REGION Network 13: Special characters — Arrows, box and block characters
   // ▄▄▄▄▄▄▄▄▄▄▄▄▄▄▄▄▄▄▄▄▄▄▄▄▄▄▄▄▄▄▄▄▄▄▄▄▄▄▄▄▄▄▄▄
   // ARROWS
   // 
   // 
   // ← Left Arrow              ⇐ Left dbl Arrow             ↩ Left Arrow Hook
   // ↑ Up Arrow               ⇑ Up dbl Arrow               ↪ Right Arrow Hook
   // → Right Arrow              ⇒ Right dbl Arrow           ⤣ North West Arrow Hook
   // ↓ Down Arrow             ⇓ Down dbl Arrow             ⤤ North East Arrow Hook
   // ↔ Left Right Arrow             ⇔ Left Right dbl Arrow          ⤥ South East Arrow Hook
   // ↕ Up Down Arrow          ⇕ Up Down dbl Arrow          ⤦ South West Arrow Hook
   // ↖ North West Arrow          ⇖ North West dbl Arrow         ↰    Up Arrow Tip Left
   // ↗ North East Arrow          ⇗ North East dbl Arrow          ↱    Up Arrow Tip Right
   // ↘ South East Arrow          ⇘ South East dbl Arrow         ↲    Down Arrow Tip Left
   // ↙ South West Arrow         ⇙    South West dbl Arrow        ↳ Down Arrow Tip Right
   // ⤡ North West & South East Arrow    ⤂ Left dbl Arrow vert Stroke       ↴ Right Arrow Corner down
   // ⤢ North East & South West Arrow    ⤃ Right dbl Arrow vert Stroke     ↵ Down Arrow Corner Left
   // ⇄ Right Arrow Over Left Arrow       ⤆ Left dbl Arrow From Bar        ↶ Anticlockwise Top Semicircle Arrow
   // ⇅ Up Arrow Left Of down Arrow        ⤇ Right dbl Arrow From Bar         ↷ Clockwise Top Semicircle Arrow
   // ⇆ Left Arrow Over Right Arrow       ⤄ Left Right dbl Arrow vert Stroke    ↺ Anticlockwise Open Circle Arrow
   // ⇇ Left Paired Arrows           ↼ Left Harpoon Barb up         ↻ Clockwise Open Circle Arrow
   // ⇈ Up Paired Arrows             ↽ Left Harpoon Barb down         ⟲ Anticlockwise Gapped Circle Arrow
   // ⇉ Right Paired Arrows         ↾ Up Harpoon Barb Right         ⟳ Clockwise Gapped Circle Arrow
   // ⇊ Down Paired Arrows           ↿ Up Harpoon Barb Left
   // ↤ Left Arrow From Bar           ⇀ Right Harpoon Barb up         ▲  Black Up Triangle 
   // ↥ Up Arrow From Bar          ⇁ Right Harpoon Barb down       ▼  Black Down Triangle
   // ↦ Right Arrow From Bar         ⇂ Down Harpoon Barb Right      ▶  Black Right Triangle
   // ↧ down Arrow From Bar        ⇃ Down Harpoon Barb Left         ◀  Black Left Triangle
   // ↨ Up Down Arrow Base         ⇋ Left Harpoon Over Right Harpoon
   // ↞ Left Two head Arrow          ⇌ Right Harpoon Over Left Harpoon
   // ↟ up Two head Arrow         ↯ Down Zigzag Arrow
   // ↠ Right Two head Arrow
   // ↡ Down Two head Arrow
   // ⤙ Left Arrow-Tail
   // ⤚ Right Arrow-Tail
   // ⤛ Left dbl Arrow-Tail    
   // ⤜ Right dbl Arrow-Tail    
   // ⤝ Left Arrow To Black Diamond    
   // ⤞ Right Arrow To Black Diamond    
   // 
   // ⟵  Long Left Arrow             ↢ Left Arrow Tail             ⌃   Up Arrowhead
   // ⟶  Long Right Arrow          ↣ Right Arrow Tail             ⌄   Down Arrowhead
   // ⟷  Long Left Right Arrow         ⤟ Left Arrow Bar To Black Diamond   ⌅   Projective
   // ⟸  Long Left dbl Arrow         ⤠ Right Arrow Bar To Black Diamond    ⌆   Perspective
   // ⟹  Long Right dbl Arrow          ⤌    Left dbl Dash Arrow         ⟰ Up Quadruple Arrow
   // ⟺  Long Left Right dbl Arrow        ⤍    Right dbl Dash Arrow         ⟱ Down Quadruple Arrow
   // ⟻  Long Left Arrow From Bar       ⤎    Left Triple Dash Arrow        ⤊ Up Triple Arrow
   // ⟼  Long Right Arrow From Bar        ⤏    Right Triple Dash Arrow         ⤋ Down Triple Arrow
   // ⟽  Long Left dbl Arrow From Bar       ⤈    Down Arrow horiz Stroke          ⤈   Down Arrow horiz Stroke
   // ⟾  Long Right dbl Arrow From Bar    ⤉    Up Arrow horiz Stroke             ⤉   Up Arrow horiz Stroke
   // 
   // 
   // 
   // ▄▄▄▄▄▄▄▄▄▄▄▄▄▄▄▄▄▄▄▄▄▄▄▄▄▄▄▄▄▄▄▄▄▄▄▄▄▄▄▄▄▄▄▄
   // BOX CHARACTERS
   // 
   // 
   // ─ Box Light horiz            ╌ Box Light dbl Dash horiz       ⋮     Vert Ellipsis
   // │ Box Light vert             ╎ Box Light dbl Dash vert        ⋯    Midline horiz Ellipsis
   // ╱ Box Light diag top Right Left      ╍ Box Heavy dbl Dash horiz       ⋰     Up Right diag Ellipsis
   // ╲ Box Light diag top Left To btm Right    ╏ Box Heavy dbl Dash vert          ⋱    Down Right diag Ellipsis
   // ╳ Box Light diag Cross          ┄ Box Light Triple Dash horiz      ╴ Box Light Left
   // ━ Box Heavy horiz             ┆ Box Light Triple Dash vert       ╵ Box Light Up
   // ┃ Box Heavy vert           ┅ Box Heavy Triple Dash horiz       ╶ Box Light Right
   // ═ Box dbl horiz               ┇ Box Heavy Triple Dash vert        ╷ Box Light Down
   // ║ Box dbl vert              ┈ Box Light Quadruple Dash horiz     ╸ Box Heavy Left
   //                       ┊ Box Light Quadruple Dash vert       ╹ Box Heavy Up
   //                       ┉ Box Heavy Quadruple Dash horiz      ╺ Box Heavy Right
   //                       ┋ Box Heavy Quadruple Dash vert     ╻ Box Heavy Down
   // 
   // ┌ Box Light Down & Right        ├ Box Light vert & Right         ─ Box Light horiz
   // └ Box Light Up & Right           ┤ Box Light vert & Left        │ Box Light vert
   // ┐ Box Light Down & Left           ┬ Box Light Down & horiz         ┼ Box Light vert & horiz
   // ┘ Box Light Up & Left          ┴ Box Light Up & horiz  
   // ┏ Box Heavy Down & Right         ┣ Box Heavy vert & Right          ━ Box Heavy horiz
   // ┗ Box Heavy Up & Right         ┫ Box Heavy vert & Left         ┃ Box Heavy vert
   // ┓ Box Heavy Down & Left         ┳ Box Heavy Down & horiz       ╋ Box Heavy vert & horiz
   // ┛ Box Heavy Up & Left        ┻ Box Heavy Up & horiz  
   //     
   // ┍ Box Down Light & Right Heavy     ┝ Box vert Light & Right Heavy      ━ Box Heavy horiz
   // ┕ Box Up Light & Right Heavy        ┥ Box vert Light & Left Heavy     │ Box Light vert
   // ┑ Box Down Light & Left Heavy     ┯ Box Down Light & horiz Heavy      ┿ Box vert Light & horiz Heavy
   // ┙ Box Up Light & Left Heavy       ┷ Box Up Light & horiz Heavy  
   // 
   // ┎ Box Down Heavy & Right Light     ┠ Box vert Heavy & Right Light      ─ Box Light horiz
   // ┖ Box Up Heavy & Right Light        ┨ Box vert Heavy & Left Light     ┃ Box Heavy vert
   // ┒ Box Down Heavy & Left Light     ┰ Box Down Heavy & horiz Light      ╂ Box vert Heavy & horiz Light
   // ┚ Box Up Heavy & Left Light       ┸ Box Up Heavy & horiz Light  
   // 
   // ┦ Box Up Heavy & Left Down Light     ┪ Box Up Light & Left Down Heavy     ╀ Box Up Heavy & Down horiz Light
   // ┶ Box Right Heavy & Left Up Light   ┹ Box Right Light & Left Up Heavy   ┾ Box Right Heavy & Left vert Light
   // ┟ Box Down Heavy & Right Up Light     ┡ Box Down Light & Right Up Heavy     ╁ Box Down Heavy & Up horiz Light
   // ┭ Box Left Heavy & Right Down Light    ┲ Box Left Light & Right Down Heavy    ┽ Box Left Heavy & Right vert Light
   //  
   // ┞ Box Up Heavy & Right Down Light     ┢ Box Up Light & Right Down Heavy     ╈ Box Up Light & Down horiz Heavy
   // ┮ Box Right Heavy & Left Down Light    ┱ Box Right Light & Left Down Heavy    ╉ Box Right Light & Left vert Heavy
   // ┧ Box Down Heavy & Left Up Light     ┩ Box Down Light & Left Up Heavy     ╇ Box Down Light & Up horiz Heavy
   // ┵ Box Left Heavy & Right Up Light      ┺ Box Left Light & Right Up Heavy   ╊ Box Left Light & Right vert Heavy
   // 
   // ╼ Box Light Left & Heavy Right                            ╄ Box Right Up Heavy & Left Down Light
   // ╽ Box Light Up & Heavy Down                            ╆ Box Right Down Heavy & Left Up Light
   // ╾ Box Heavy Left & Light Right                            ╅ Box Left Down Heavy & Right Up Light
   // ╿ Box Heavy Up & Light Down                            ╃ Box Left Up Heavy & Right Down Light
   // 
   // ╔ Box dbl Down & Right         ╠ Box dbl vert & Right         ═ Box dbl horiz
   // ╚ Box dbl Up & Right           ╣ Box dbl vert & Left           ║ Box dbl vert
   // ╗ Box dbl Down & Left        ╦ Box dbl Down & horiz         ╬ Box dbl vert & horiz
   // ╝ Box dbl Up & Left          ╩ Box dbl Up & horiz  
   //  
   // ╒ Box Down Single & Right dbl     ╞ Box vert Single & Right dbl      ═ Box dbl horiz
   // ╘ Box Up Single & Right dbl        ╡ Box vert Single & Left dbl        │ Box Light vert
   // ╕ Box Down Single & Left dbl        ╤ Box Down Single & horiz dbl      ╪ Box vert Single & horiz dbl
   // ╛ Box Up Single & Left dbl       ╧ Box Up Single & horiz dbl  
   // 
   // ╓ Box Down dbl & Right Single     ╟ Box vert dbl & Right Single      ─ Box Light horiz
   // ╙ Box Up dbl & Right Single        ╢ Box vert dbl & Left Single        ║ Box dbl vert
   // ╖ Box Down dbl & Left Single        ╥ Box Down dbl & horiz Single      ╫ Box vert dbl & horiz Single
   // ╜ Box Up dbl & Left Single       ╨ Box Up dbl & horiz Single  
   // 
   // 
   // 
   // ▄▄▄▄▄▄▄▄▄▄▄▄▄▄▄▄▄▄▄▄▄▄▄▄▄▄▄▄▄▄▄▄▄▄▄▄▄▄▄▄▄▄▄▄
   // BLOCK CHARACTERS
   // 
   // 
   // ▀ Top Half Block             ❘    Light vert Bar              ❘ ❘     En Space
   // ▄ Btm Half Block            ❙    Medium vert Bar           ❘ ❘   Em Space
   // ▐ Right Half Block          ❚   Heavy vert Bar  
   // ▌ Left Half Block    
   // 
   // ▔ Top One Eighth Block        ▉ Left Seven Eighths Block
   // ▁ Btm One Eighth Block          ▊ Left Three Quarters Block
   // ▂ Btm One Quarter Block        ▋ Left Five Eighths Block
   // ▃ Btm Three Eighths Block      ▌ Left Half Block
   // ▄ Btm Half Block            ▍ Left Three Eighths Block
   // ▅ Btm Five Eighths Block         ▎ Left One Quarter Block
   // ▆ Btm Three Quarters Block       ▏ Left One Eighth Block
   // ▇ Btm Seven Eighths Block        ▕ Right One Eighth Block
   // █ Full Block
   // ░ Light Shade
   // ▒ Medium Shade    
   // ▓ Dark Shade    
   // 
   // 
   // ██████████████ █ █ █ █  END   █ █ █ █ ██████████████
END_REGION

REGION Network 14: Special characters — Currency, punctuation and full-width characters
   // ▄▄▄▄▄▄▄▄▄▄▄▄▄▄▄▄▄▄▄▄▄▄▄▄▄▄▄▄▄▄▄▄▄▄▄▄▄▄▄▄▄▄▄▄
   // CURRENCY
   // 
   // 
   // ₳   Austral Sign             €   Euro Sign              ₦  Naira Sign
   // ₵   Cedi Sign               ₠  Euro-Currency Sign          ₪  New Shekel Sign
   // ¢   Cent Sign              ₣  French Franc Sign           ₧   Peseta Sign
   // ₡   Colon Sign               ₰   German Penny Sign           ₱   Peso Sign
   // ₢   Cruzeiro Sign           ₲   Guarani Sign              £  Pound Sign
   // ¤  Currency Sign             ₴   Hryvnia Sign            ₨    Rupee Sign
   // $   Dollar Sign            ₭   Kip Sign              ₮   Tugrik Sign
   // ₫   Dong Sign             ₤   Lira Sign             ₩  Won Sign
   // ₯ Drachma Sign            ₥  Mill Sign              ¥   Yen Sign
   // 
   // 
   // 
   // ▄▄▄▄▄▄▄▄▄▄▄▄▄▄▄▄▄▄▄▄▄▄▄▄▄▄▄▄▄▄▄▄▄▄▄▄▄▄▄▄▄▄▄▄
   // PUNCTUATION AND COMMON SYMBOLS
   // 
   // 
   // #  Hash Sign             "   Quote                 §   Section Sign
   // $   Dollar Sign            “    Left dbl quote             ¶   Pilcrow Sign
   // %  Percent Sign            ”    Right dbl quote
   // &   Ampersand             '    Apostrophe  
   // *   Asterisk              ‘    Left Single quote          †   Dagger
   // ~   Tilde                 ’    Right Single quote           ‡   Dbl Dagger
   // +   Plus Sign               ‹    Single Left Angle quote       •   Bullet
   // -    Hyphen/minus            ›    Single Right Angle quote        ·    Middle Dot
   // =   Equals Sign                                ‣   Triangular Bullet
   // <   Less-Than Sign           ´   Acute Accent              ⁃    Hyphen Bullet
   // >   Greater-Than Sign           `   Grave Accent
   // (    Left Parenthesis
   // )    Right Parenthesis            ©  Copyright Sign           ⁎   Low Asterisk
   // [    Left Square Bracket           ®  Registered Sign  
   // ]    Right Square Bracket         ℀  Account Of               ․    One Dot Leader
   // {   Left Curly Bracket          ℁  Addressed To The Subject      ‥   Two Dot Leader
   // }   Right Curly Bracket          ℂ  Dbl-Struck Capital C           …  Horiz Ellipsis
   // 〈    Left Angle Bracket           ℄   Centre Line Symbol  
   // 〉    Right Angle Bracket            ℅  Care Of               ※  Reference Mark
   // ⁅    Left Square Bracket Quill        ℗  Sound Recording Copyright       ‼   Dbl Exclamation Mark
   // ⁆    Right Square Bracket Quill      ™  Trade Mark Sign            ‽   Interrobang
   // ,    Comma                                 ⁇  Dbl Question Mark
   // .    Full Stop                                   ⁈   Question Exclamation Mark
   // :    Colon                                  ⁉  Exclamation Question Mark
   // ;    Semicolon    
   // !    Exclamation Mark            ⁑   Two Asterisks Aligned vertically     |    Vert Line
   // ?   Question Mark           ⁂   Asterism               ¦    Broken Bar
   // @  Commercial At                              ‖    Dbl vert Line
   // ^   Circumflex Accent            ⁀  Character Tie              ‗   Dbl Low Line
   // /    Solidus               ‿  Undertie             ⁞    Vert Four Dots
   // \    Reverse Solidus            ⁐  Close Up
   // _   Underscore
   // ― Horiz Bar    
   // ¯   Macron
   // ‾   Overline
   // 
   // 
   // 
   // ▄▄▄▄▄▄▄▄▄▄▄▄▄▄▄▄▄▄▄▄▄▄▄▄▄▄▄▄▄▄▄▄▄▄▄▄▄▄▄▄▄▄▄▄
   // NON-PROPORTIONAL (FULL-WIDTH) LETTERS
   // 
   // 
   // Ａ Fullwidth Capital Letter A        ａ Fullwidth Small Letter A       ＂ Fullwidth quote
   // Ｂ Fullwidth Capital Letter B        ｂ Fullwidth Small Letter B       ＇ Fullwidth Apostrophe
   // Ｃ Fullwidth Capital Letter C        ｃ Fullwidth Small Letter C       ＃ Fullwidth Number Sign
   // Ｄ Fullwidth Capital Letter D       ｄ Fullwidth Small Letter D       ＄ Fullwidth Dollar Sign
   // Ｅ Fullwidth Capital Letter E        ｅ Fullwidth Small Letter E       ％ Fullwidth Percent Sign
   // Ｆ Fullwidth Capital Letter F        ｆ Fullwidth Small Letter F       ＆ Fullwidth Ampers&
   // Ｇ Fullwidth Capital Letter G       ｇ Fullwidth Small Letter G       ＊ Fullwidth Asterisk
   // Ｈ Fullwidth Capital Letter H       ｈ Fullwidth Small Letter H          ～ Fullwidth Tilde
   // Ｉ Fullwidth Capital Letter I         ｉ Fullwidth Small Letter I        ＋ Fullwidth Plus Sign
   // Ｊ Fullwidth Capital Letter J         ｊ Fullwidth Small Letter J        － Fullwidth Hyphen-Minus
   // Ｋ Fullwidth Capital Letter K        ｋ Fullwidth Small Letter K       ＝ Fullwidth Equals Sign
   // Ｌ Fullwidth Capital Letter L        ｌ Fullwidth Small Letter L       ＜ Fullwidth Less-Than Sign
   // Ｍ Fullwidth Capital Letter M       ｍ Fullwidth Small Letter M         ＞ Fullwidth Greater-Than Sign
   // Ｎ Fullwidth Capital Letter N       ｎ Fullwidth Small Letter N          （ Fullwidth Left Parenthesis
   // Ｏ Fullwidth Capital Letter O       ｏ Fullwidth Small Letter O       ） Fullwidth Right Parenthesis
   // Ｐ Fullwidth Capital Letter P        ｐ Fullwidth Small Letter P       ［ Fullwidth Left Square Bracket
   // Ｑ Fullwidth Capital Letter Q       ｑ Fullwidth Small Letter Q         ］ Fullwidth Right Square Bracket
   // Ｒ Fullwidth Capital Letter R        ｒ Fullwidth Small Letter R       ｛ Fullwidth Left Curly Bracket
   // Ｓ Fullwidth Capital Letter S        ｓ Fullwidth Small Letter S       ｝ Fullwidth Right Curly Bracket
   // Ｔ Fullwidth Capital Letter T        ｔ Fullwidth Small Letter T        ， Fullwidth Comma
   // Ｕ Fullwidth Capital Letter U       ｕ Fullwidth Small Letter U       ． Fullwidth Full Stop
   // Ｖ Fullwidth Capital Letter V        ｖ Fullwidth Small Letter V       ： Fullwidth Colon
   // Ｗ Fullwidth Capital Letter W       ｗ Fullwidth Small Letter W         ； Fullwidth Semicolon
   // Ｘ Fullwidth Capital Letter X        ｘ Fullwidth Small Letter X       ！ Fullwidth Exclamation Mark
   // Ｙ Fullwidth Capital Letter Y        ｙ Fullwidth Small Letter Y       ？ Fullwidth Question Mark
   // Ｚ Fullwidth Capital Letter Z        ｚ Fullwidth Small Letter Z       ＠ Fullwidth Commercial At
   //                                         ＾ Fullwidth Circumflex Accent
   // ０ Fullwidth Digit Zero         ５ Fullwidth Digit Five          ／ Fullwidth Solidus
   // １ Fullwidth Digit One         ６ Fullwidth Digit Six         ＼ Fullwidth Reverse Solidus
   // ２ Fullwidth Digit Two          ７ Fullwidth Digit Seven         ＿ Fullwidth Low Line
   // ３ Fullwidth Digit Three          ８ Fullwidth Digit Eight           ｜ Fullwidth vert Line
   // ４ Fullwidth Digit Four         ９ Fullwidth Digit Nine         ❘ ❘   Fullwidth space    
   // 
   // 
   // ██████████████ █ █ █ █  END   █ █ █ █ ██████████████
END_REGION

REGION Network 15: Special characters — Greek, indexing characters and Roman numerals
   // ▄▄▄▄▄▄▄▄▄▄▄▄▄▄▄▄▄▄▄▄▄▄▄▄▄▄▄▄▄▄▄▄▄▄▄▄▄▄▄▄▄▄▄▄
   // GREEK CHARACTERS
   // 
   // 
   // Α  Greek Capital Letter Alpha        α   Greek Small Letter Alpha
   // Β   Greek Capital Letter Beta       β   Greek Small Letter Beta
   // Γ   Greek Capital Letter Gamma       γ   Greek Small Letter Gamma
   // Δ  Greek Capital Letter Delta      δ   Greek Small Letter Delta
   // Ε   Greek Capital Letter Epsilon     ε   Greek Small Letter Epsilon
   // Ζ   Greek Capital Letter Zeta       ζ   Greek Small Letter Zeta
   // Η  Greek Capital Letter Eta       η   Greek Small Letter Eta
   // Θ  Greek Capital Letter Theta      θ   Greek Small Letter Theta
   // Ι    Greek Capital Letter Iota         ι    Greek Small Letter Iota
   // Κ   Greek Capital Letter Kappa       κ   Greek Small Letter Kappa
   // Λ   Greek Capital Letter Lambda       λ   Greek Small Letter Lambda
   // Μ  Greek Capital Letter Mu       μ   Greek Small Letter Mu
   // Ν  Greek Capital Letter Nu        ν   Greek Small Letter Nu
   // Ξ   Greek Capital Letter Xi         ξ   Greek Small Letter Xi
   // Ο  Greek Capital Letter Omicron      ο   Greek Small Letter Omicron
   // Π  Greek Capital Letter Pi          π   Greek Small Letter Pi
   // Ρ   Greek Capital Letter Rho      ρ   Greek Small Letter Rho
   // Σ   Greek Capital Letter Sigma       ς   Greek Small Letter Final Sigma
   //                       σ   Greek Small Letter Sigma
   // Τ   Greek Capital Letter Tau         τ   Greek Small Letter Tau
   // Υ   Greek Capital Letter Upsilon     υ   Greek Small Letter Upsilon
   // Φ  Greek Capital Letter Phi       φ  Greek Small Letter Phi
   // Χ   Greek Capital Letter Chi       χ   Greek Small Letter Chi
   // Ψ  Greek Capital Letter Psi        ψ  Greek Small Letter Psi
   // 
   // 
   // 
   // ▄▄▄▄▄▄▄▄▄▄▄▄▄▄▄▄▄▄▄▄▄▄▄▄▄▄▄▄▄▄▄▄▄▄▄▄▄▄▄▄▄▄▄▄
   // INDEXING CHARACTERS  (all characters are 1 EM wide)
   // 
   // 
   // ① Circled One              ⑴ Bracketed One           ⒈ One Full Stop
   // ② Circled Two              ⑵ Bracketed Two           ⒉ Two Full Stop
   // ③ Circled Three              ⑶ Bracketed Three           ⒊ Three Full Stop
   // ④ Circled Four             ⑷ Bracketed Four             ⒋ Four Full Stop
   // ⑤ Circled Five              ⑸ Bracketed Five           ⒌ Five Full Stop
   // ⑥ Circled Six             ⑹ Bracketed Six             ⒍ Six Full Stop
   // ⑦ Circled Seven             ⑺ Bracketed Seven          ⒎ Seven Full Stop
   // ⑧ Circled Eight            ⑻ Bracketed Eight            ⒏ Eight Full Stop
   // ⑨ Circled Nine             ⑼ Bracketed Nine          ⒐ Nine Full Stop
   // ⑩ Circled Ten            ⑽ Bracketed Ten            ⒑ Ten Full Stop
   // ⑪ Circled Eleven            ⑾ Bracketed Eleven         ⒒ Eleven Full Stop
   // ⑫ Circled Twelve            ⑿ Bracketed Twelve         ⒓ Twelve Full Stop
   // ⑬ Circled Thirteen             ⒀ Bracketed Thirteen          ⒔ Thirteen Full Stop
   // ⑭ Circled Fourteen           ⒁ Bracketed Fourteen        ⒕ Fourteen Full Stop
   // ⑮ Circled Fifteen            ⒂ Bracketed Fifteen         ⒖ Fifteen Full Stop
   // ⑯ Circled Sixteen           ⒃ Bracketed Sixteen           ⒗ Sixteen Full Stop
   // ⑰ Circled Seventeen           ⒄ Bracketed Seventeen        ⒘ Seventeen Full Stop
   // ⑱ Circled Eighteen           ⒅ Bracketed Eighteen        ⒙ Eighteen Full Stop
   // ⑲ Circled Nineteen           ⒆ Bracketed Nineteen           ⒚ Nineteen Full Stop
   // ⑳ Circled Twenty            ⒇ Bracketed Twenty         ⒛ Twenty Full Stop
   // 
   // 
   // 
   // ▄▄▄▄▄▄▄▄▄▄▄▄▄▄▄▄▄▄▄▄▄▄▄▄▄▄▄▄▄▄▄▄▄▄▄▄▄▄▄▄▄▄▄▄
   // ROMAN NUMERALS
   // 
   // 
   // Ⅰ    Roman num One          ⅰ    Small Roman num One
   // Ⅱ   Roman num Two           ⅱ   Small Roman num Two
   // Ⅲ  Roman num Three           ⅲ  Small Roman num Three
   // Ⅳ  Roman num Four          ⅳ  Small Roman num Four
   // Ⅴ   Roman num Five          ⅴ   Small Roman num Five
   // Ⅵ  Roman num Six             ⅵ  Small Roman num Six
   // Ⅶ Roman num Seven         ⅶ    Small Roman num Seven
   // Ⅷ    Roman num Eight           ⅷ   Small Roman num Eight
   // Ⅸ  Roman num Nine            ⅸ  Small Roman num Nine
   // Ⅹ   Roman num Ten           ⅹ   Small Roman num Ten
   // Ⅺ  Roman num Eleven           ⅺ  Small Roman num Eleven
   // Ⅻ Roman num Twelve           ⅻ  Small Roman num Twelve
   // Ⅼ   Roman num Fifty           ⅼ    Small Roman num Fifty
   // Ⅽ   Roman num One Hundred        ⅽ   Small Roman num One Hundred
   // Ⅾ  Roman num Five Hundred      ⅾ   Small Roman num Five Hundred
   // Ⅿ  Roman num One Thousand      ⅿ     Small Roman num One Thousand    
   // 
   // 
   // ████████████████████ END    ████████████████████
END_REGION

REGION Network 16: Special characters — Mathematical operators (including vulgar fractions)
   // ▄▄▄▄▄▄▄▄▄▄▄▄▄▄▄▄▄▄▄▄▄▄▄▄▄▄▄▄▄▄▄▄▄▄▄▄▄▄▄▄▄▄▄▄
   // MATHEMATICAL OPERATORS
   // 
   // 
   // ×   Multiplication Sign          ¹   Superscript One           ∅  Empty Set
   // ÷   Division Sign              ²   Superscript Two            ∈  Element Of
   // +   Plus sign                ³   Superscript Three         ∉  Not An Element Of
   // −   Minus Sign            ½  Vulgar Fraction One Half         ∊   Small Element Of
   // ⁒   Commercial Minus Sign       ⅓  Vulgar Fraction One Third       ∋  Contains As Member
   // ±   Plus-Minus Sign             ⅔  Vulgar Fraction Two Thirds      ∌  Does Not Contain As Member
   // ∓   Minus-Or-Plus Sign          ¼  Vulgar Fraction One Quarter        ∍   Small Contains As Member
   // ≤   Less-Than Or Equal To       ¾  Vulgar Fraction Three Quarters      ∩   Intersection
   // ≥   Greater-Than Or Equal To        ⅕  Vulgar Fraction One Fifth        ∪   Union
   // ≪  Much Less-Than            ⅖  Vulgar Fraction Two Fifths       ⊂  Subset Of
   // ≫  Much Greater-Than          ⅗  Vulgar Fraction Three Fifths       ⊃  Superset Of
   // √  Square Root             ⅘  Vulgar Fraction Four Fifths      ⊄  Not A Subset Of
   // ∛  Cube Root             ⅙  Vulgar Fraction One Sixth       ⊅  Not A Superset Of
   // ∜  Fourth Root              ⅚  Vulgar Fraction Five Sixths        ⊆  Subset Of Or Equal To
   // ∝  Proportional To           ⅛  Vulgar Fraction One Eighth       ⊇  Superset Of Or Equal To
   // ∞  Infinity              ⅜  Vulgar Fraction Three Eighths      ⊈  not A Subset Of Nor Equal To
   // °   Degree Sign            ⅝  Vulgar Fraction Five Eighths     ⊉  not A Superset Of Nor Equal To
   // µ   Micro Sign             ⅞  Vulgar Fraction Seven Eighths    ⊊  Subset Of Not Equal To
   // ‰   Per Mille Sign              ⅟   Fraction Numerator One         ⊋  Superset Of Not Equal To
   // ‱  Per Ten Thousand& Sign          ⁄    Fraction Slash            ⊌   Multiset
   // ∀  For All                                    ⊍   Multiset Multiplication
   // ∁   Complement                                 ⊎   Multiset Union
   // ∂   Partial Differential                              ⊏  Square Image Of
   // ∃   There Exists                                ⊐  Square Original Of
   // ∄   There Does Not Exist          ∆   Increment             ⊑  Square Image Of Or Equal To
   // ∴    Therefore               ∇  Nabla               ⊒  Square Original Of Or Equal To
   // ∵    Because                                   ⊓  Square Cap
   // ∶   Ratio                                   ⊔  Square Cup
   // ∷  Proportion    
   // ∿  Sine Wave    
   //      
   // ∥   Parallel To             ∫    Integral               ⌠    Top Half Integral
   // ∦   Not Parallel To            ∬    Dbl Integral              ⌡    Bottom Half Integral
   // ∟ Right Angle              ∭   Triple Integral             ❲   Light Left Shell Bracket 
   // ⊾  Right Angle Arc           ∮   Contour Integral           ❳   Light Right Shell Bracket 
   // ⊿  Right Triangle             ∯    Surface Integral            ⟪   Maths Left dbl Angle Bracket
   // ∠  Angle               ∰   Volume Integral            ⟫   Maths Right dbl Angle Bracket
   // ∡  Measured Angle           ∱   Clockwise Integral           ⟬   Maths Left White Shell Bracket
   // ∢  Spherical Angle            ∲   Clockwise Contour Integral       ⟭   Maths Right White Shell Bracket
   // ⌒    Arc                 ∳   Anticlockwise Contour Integral
   // ⌓    Segment    
   // ⌔     Sector    
   // 
   // ≃   Asymptotically Equal To       ⊕    Circled Plus              ′    Prime
   // ≄   Not Asymptotically Equal To      ⊖    Circled Minus              ″    Dbl Prime
   // ≅   Approx Equal To            ⊗    Circled Times              ‴   Triple Prime
   // ≆   Approx But Not Actually Equal To    ⊘    Circled Division Slash        ⁗   Quadruple Prime
   // ≇   Not approx Nor Actually Equal To   ⊙    Circled Dot Operator          ‵    Reversed Prime
   // ≈   Almost Equal To            ⊚    Circled Ring Operator        ‶    Reversed dbl Prime
   // ≉  Not Almost Equal To          ⊛    Circled Asterisk Operator        ‷   Reversed Triple Prime
   // ≊   Almost Equal Or Equal To       ⊜    Circled Equals
   // ≋   Triple Tilde             ⊝    Circled Dash
   // ≌   All Equal To              ⊞    Squared Plus
   // ≍  Equivalent To             ⊟    Squared Minus
   // ≡   Identical To              ⊠    Squared Times
   // ≢   Not Identical To             ⊡    Squared Dot Operator
   //      
   // ∧  Logical &               ⊢  Right Tack              °   Degree Sign
   // ∨  Logical Or             ⊣  Left Tack                ℃    Degree Celsius
   // ⊻  Xor                 ⊤  Down Tack               ℉    Degree Fahrenheit
   // ⊼  Nand                ⊥  Up Tack                Ω    Ohm Sign    
   // 
   // 
   // ██████████████ █ █ █ █  END   █ █ █ █ ██████████████
END_REGION

REGION Network 17: Special characters — Geometrical and ornamental characters
   // ▄▄▄▄▄▄▄▄▄▄▄▄▄▄▄▄▄▄▄▄▄▄▄▄▄▄▄▄▄▄▄▄▄▄▄▄▄▄▄▄▄▄▄▄
   // GEOMETRICAL CHARACTERS
   // 
   // 
   // ⌉    Right Ceiling            ▬  Black Rectangle            ▭  White Rectangle
   // ⌋    Right Floor                ▮   Black vert Rectangle          ▯   White vert Rectangle
   // ⌈    Left Ceiling               ▰  Black Parallelogram           ▱  White Parallelogram
   // ⌊    Left Floor               ◆  Black Diamond             ◇ White Diamond
   // ⌝   Top Right Corner 
   // ⌟   Bottom Right Corner          ◈  Diamond with Diamond          ◊  Lozenge
   // ⌜   Top Left Corner           ▲  Black Up Triangle             △  White Up Triangle
   // ⌞   Bottom Left Corner          ▶  Black Right Triangle         ▷  White Right Triangle
   // ◝ Top Right quad Circular Arc        ▼  Black Down Triangle          ▽ White Down Triangle
   // ◞ Btm Right quad Circular Arc       ◀  Black Left Triangle           ◁  White Left Triangle
   // ◜ Top Left quad Circular Arc       ▴   Black Up Small Triangle       ▵   White Up Small Triangle
   // ◟ Btm Left quad Circular Arc      ▸   Black Right Small Triangle      ▹   White Right Small Triangle
   // ◘ Inv Bullet               ▾   Black Down Small Triangle     ▿   White Down Small Triangle
   // ◙ Inv White Circle             ◂   Black Left Small Triangle         ◃   White Left Small Triangle
   // ◚ Top Half inv White Circle       ►  Black Right Pointer          ▻  White Right Pointer
   // ◛ Btm Half inv White Circle      ◄  Black Left Pointer          ◅  White Left Pointer
   //      
   // ◻  White Medium Square       ◼  Black Medium Square          ⬔    Square top Right diag Half Black
   // □  White Square              ■  Black Square           ⬕    Square btm Left diag Half Black
   // ◽   White Medium Small Square     ◾   Black Medium Small Square     ⬖    Diamond Left Half Black
   // ▫  White Small Square           ▪  Black Small Square         ⬗    Diamond Right Half Black
   // ▣  Square with Square                              ⬘    Diamond Top Half Black
   // ◉  Fisheye                                  ⬙    Diamond Bottom Half Black
   // ○  White Circle              ●  Black Circle              ◪  Square btm Right diag Half Black
   // ◌  Dotted Circle              ◍  Circle vert Fill              ◫  White Square vert Bisecting Line
   // ◯ Large Circle             ◎ Bullseye              ◬  White Up Triangle Dot
   // ▢  White Square Rounded Corners                        ◭  Up Triangle Left Black
   // ▤  Square horiz Fill                               ◮  Up Triangle Right Black
   // ▥  Square vert Fill                                ◐  Circle Left Half Black
   // ▦  Square Orthogonal Crosshatch Fill   ◖   Left Half Black Circle          ◑  Circle Right Half Black
   // ▧  Square top Left To btm Right Fill     ◗   Right Half Black Circle        ◒  Circle btm Half Black
   // ▨  Square top Right To btm Left Fill                       ◓  Circle top Half Black
   // ▩  Square diag Crosshatch Fill    
   //      
   // ◸    Top Left Triangle                                     ◰    White Square top Left quad
   // ◹    Top Right Triangle                               ◱    White Square btm Left quad
   // ◿    Btm Right Triangle                              ◲    White Square btm Right quad
   // ◺    Btm Left Triangle                                ◳    White Square top Right quad
   // ⧖  White Hourglass           ⧗  Black Hourglass            ◴    White Circle top Left quad
   // ⋈  Bowtie                                         ◵    White Circle btm Left quad
   // 
   // 
   // 
   // ▄▄▄▄▄▄▄▄▄▄▄▄▄▄▄▄▄▄▄▄▄▄▄▄▄▄▄▄▄▄▄▄▄▄▄▄▄▄▄▄▄▄▄▄
   // ORNAMENTAL CHARACTERS
   // 
   // 
   // ⌂  House              ☣  Biohazard Sign           ♚  Black Chess King
   // ⌕  Telephone Recorder           ☤  Caduceus              ♛  Black Chess Queen
   // ⌖   Position Indicator            ☥  Ankh                 ♜  Black Chess Rook
   // ⌗    Viewdata Square          ☮    Peace Symbol            ♝  Black Chess Bishop
   // ⌘    Place Of Interest Sign        ☯ Yin Yang                ♞  Black Chess Knight
   // ⌚     Watch               ☰    Trigram For Heaven           ♟  Black Chess Pawn
   // ⌛  Hourglass             ☱    Trigram For Lake           ♠  Black Spade Suit
   // ⌢  Frown                  ☲    Trigram For Fire             ♡  White Heart Suit
   // ⌣  Smile               ☳    Trigram For Thunder           ♢  White Diamond Suit
   // ⌥  Option Key            ☴    Trigram For Wind           ♣    Black Club Suit
   // ⌦   Erase To The Right           ☵    Trigram For Water            ♤  White Spade Suit
   // ⌧    X In A Rectangle Box          ☶    Trigram For Mountain           ♥  Black Heart Suit
   // ⌨  Keyboard               ☷    Trigram For Earth          ♦  Black Diamond Suit
   // ⌫   Erase To The Left          ☸ Wheel Of Dharma            ♧    White Club Suit
   //                       ☹  White Frowning Face         ♨    Hot Springs
   //                       ☺  White Smiling Face         ♩  Quarter Note
   //                       ☻  Black Smiling Face          ♪  Eighth Note
   // ☀  Black Sun Rays              ☼    White Sun Rays           ♫  Beamed Eighth Notes
   // ☁     Cloud               ☽  First Quarter Moon          ♬  Beamed Sixteenth Notes
   // ☂     Umbrella               ☾  Last Quarter Moon          ♭ Music Flat Sign
   // ☃  Snowman             ☿  Mercury               ♮  Music Natural Sign
   // ☄  Comet                 ♀  Female Sign               ♯ Music Sharp Sign
   // ★  Black Star              ♁  Earth                ⚀ Die Face-1
   // ☆ White Star             ♂    Male Sign              ⚁ Die Face-2
   // ☇   Lightning               ♃  Jupiter                 ⚂ Die Face-3
   // ☈  Thunderstorm            ♄  Saturn                 ⚃ Die Face-4
   // ☉    Sun                ♅  Uranus                ⚄ Die Face-5
   // ☊ Ascending Node           ♆   Neptune             ⚅ Die Face-6
   // ☋ Descending Node           ♇  Pluto                 ⚆ White Circle Dot Right
   // ☌  Conjunction             ♈   Aries                 ⚇ White Circle Two Dots
   // ☍    Opposition               ♉   Taurus                 ⚈ Black Circle White Dot Right
   // ☎   Black Telephone           ♊ Gemini               ⚉ Black Circle Two White Dots
   // ☏   White Telephone           ♋   Cancer                ⚠  Warning Sign
   // ☐  Ballot Box              ♌ Leo                ✁   Top Blade Scissors
   // ☑  Ballot Box Check           ♍ Virgo                ✂   Black Scissors
   // ☒  Ballot Box X              ♎    Libra                 ✃   Btm Blade Scissors
   // ☓   Saltire              ♏    Scorpius             ✄   White Scissors
   //                       ♐ Sagittarius               
   // ☚    Black Left point Index        ♑   Capricorn              ✆    Telephone Location Sign
   // ☛    Black Right point Index         ♒   Aquarius                ✇  Tape Drive
   // ☜    White Left point Index        ♓    Pisces                 ✈  Airplane
   // ☝  White Up point Index          ♔  White Chess King          ✉  Envelope
   // ☞    White Right point Index         ♕  White Chess Queen           ✍ Writing H&
   // ☟  White Down point Index       ♖  White Chess Rook         ✎   Btm Right Pencil
   // ☠ Skull & Crossbones         ♗  White Chess Bishop           ✏   Pencil
   // ☡  Caution Sign            ♘  White Chess Knight         ✐   Top Right Pencil
   // ☢    Radioactive Sign           ♙  White Chess Pawn           ✓  Check Mark
   // ✔    Heavy Check Mark           ✬    Black Centre White Star        ❂  Circled Open Centre Eight point Star
   // ✕  Multiplication X          ✭    Outlined Black Star         ❃  Heavy Teardrop Pinwheel Asterisk
   // ✖  Heavy Multiplication X       ✮    Heavy Outlined Black Star      ❄  Snowflake
   // ✗  Ballot X               ✯    Pinwheel Star             ❅  Tight Trifoliate Snowflake
   // ✘  Heavy Ballot X            ✰    Shadowed White Star        ❆  Heavy Chevron Snowflake
   // ✚  Heavy Greek Cross          ✱  Heavy Asterisk           ❇  Sparkle
   // ✛  Open Centre Cross          ✲  Open Centre Asterisk        ❈  Heavy Sparkle
   // ✜  Heavy Open Centre Cross       ✳  Eight Spoked Asterisk          ❉  Balloon Asterisk
   // ✝   Latin Cross               ✴  Eight point Black Star        ❊  Eight Teardrop Asterisk
   // ✞  Shadowed White Latin Cross       ✵  Eight point Pinwheel Star       ❋  Heavy Eight Teardrop Asterisk
   // ✟   Outlined Latin Cross          ✶  Six point Black Star         ❍    Shadowed White Circle
   // ✠  Maltese Cross            ✷  Eight point Rectilinear Black Star   ❏  Btm Right Shadowed White Square
   // ✡  Star Of David           ✸  Heavy Eight point Black Star     ❐  Top Right Shadowed White Square
   // ✢  Four Teardrop Asterisk         ✹  Twelve point Black Star        ❑  Btm Right Shadowed White Square
   // ✣  Four Balloon Asterisk         ✺  Sixteen point Asterisk        ❒  Top Right Shadowed White Square
   // ✤  Heavy Four Balloon Asterisk      ✻  Teardrop Asterisk            ❖  Black Diamond Minus White X
   // ✥  Four Club Asterisk           ✼  Open Centre Teardrop Asterisk      
   // ✦  Black Four point Star         ✽  Heavy Teardrop Asterisk         ❛   Heavy Single Turned Comma quote 
   // ✧  White Four point Star         ✾  Six Petalled Black & White Florette    ❜   Heavy Single Comma quote 
   // ✩    Stress Outlined White Star        ✿  Black Florette             ❝  Heavy dbl Turned Comma quote 
   // ✪  Circled White Star            ❀  White Florette             ❞  Heavy dbl Comma quote 
   // ✫    Open Centre Black Star        ❁  Eight Petalled Black Florette     
   // 
   // 
   // ██████████████ █ █ █ █  END   █ █ █ █ ██████████████
END_REGION

REGION Network 18: Special characters — Common character widths and additional whitespace characters
   // ▀▀▀▀▀▀▀▀▀▀▀▀▀▀▀▀▀▀▀▀▀▀▀▀▀▀▀▀▀▀▀▀▀▀▀▀▀▀▀▀▀▀▀▀
   // 
   // TITLE:    COMMON CHARACTER WIDTHS AND ADDITIONAL WHITESPACE CHARACTERS
   // 
   // ▄▄▄▄▄▄▄▄▄▄▄▄▄▄▄▄▄▄▄▄▄▄▄▄▄▄▄▄▄▄▄▄▄▄▄▄▄▄▄▄▄▄▄▄
   // 
   // 
   // 
   // This section contains a list of the alphanumeric characters and common punctuation in terms of
   // character width (thinnest first).
   // 
   // The average character widths for each group are based on the frequency of letter usage in 
   // standard (British) English.
   // 
   // The additional whitespace characters complete the set of TIA Portal whitespace characters, these
   // are included for completeness, but duplicate the widths of the standard whitespace characters 
   // listed in previous sections.
   // 
   // 
   // 
   // ▄▄▄▄▄▄▄▄▄▄▄▄▄▄▄▄▄▄▄▄▄▄▄▄▄▄▄▄▄▄▄▄▄▄▄▄▄▄▄▄▄▄▄▄
   // NORMAL CHARACTERS BY WIDTH
   // 
   // 
   // ▐I▌1sp
   // ▐J▌1⅓ sp
   // ▐T▌1⅔ SP
   // ▐F▌2 sp
   // ▐L▌2 sp
   // ▐P▌2 sp
   // ▐R▌2 sp
   // ▐A▌2⅓ SP
   // ▐B▌2⅓ SP
   // ▐C▌2⅓ SP
   // ▐E▌2⅓3 SP
   // ▐K▌2⅓ SP
   // ▐S▌2⅓ SP
   // ▐V▌2⅓ SP
   // ▐X▌2⅓ SP
   // ▐Y▌2⅓ SP
   // ▐Z▌2⅓ SP
   // ▐D▌2⅔ sp
   // ▐G▌2⅔ sp
   // ▐H▌2⅔ sp
   // ▐N▌2⅔ sp
   // ▐U▌2⅔ sp
   // ▐M▌3 sp
   // ▐O▌3 sp
   // ▐Q▌3 sp
   // ▐W▌3 sp
   // Upper avg. (based on frequency and width) = 2.25 normal spaces
   // 
   // ▐f▌1 sp
   // ▐i▌1 sp
   // ▐j▌1 sp
   // ▐l▌1 sp
   // ▐r▌1⅓ sp
   // ▐t▌1⅓ sp
   // ▐x▌1⅔ sp
   // ▐y▌1⅔ sp
   // ▐z▌1⅔ sp
   // ▐c▌2 sp
   // ▐k▌2 sp
   // ▐s▌2 sp
   // ▐v▌2 sp
   // ▐a▌2⅓ sp
   // ▐b▌2⅓ sp
   // ▐d▌2⅓ sp
   // ▐e▌2⅓ sp
   // ▐g▌2⅓ sp
   // ▐h▌2⅓ sp
   // ▐n▌2⅓ sp
   // ▐o▌2⅓ sp
   // ▐p▌2⅓ sp
   // ▐q▌2⅓ sp
   // ▐u▌2⅓ sp
   // ▐w▌3 sp
   // ▐m▌3⅔ sp
   // Lower avg. (based on frequency and width) = 2.00 normal spaces
   // 
   // ▐0▌2⅓ sp
   // ▐1▌2⅓ sp
   // ▐2▌2⅓ sp
   // ▐3▌2⅓ sp
   // ▐4▌2⅓ sp
   // ▐5▌2⅓ sp
   // ▐6▌2⅓ sp
   // ▐7▌2⅓ sp
   // ▐8▌2⅓ sp
   // ▐9▌2⅓ sp
   // Numbers = 2.33 sp
   // 
   // ▐!▌1 sp
   // ▐'▌1 sp
   // ▐,▌1 sp
   // ▐-▌1 sp
   // ▐.▌1 sp
   // ▐/▌1 sp
   // ▐\▌1 sp
   // ▐|▌1 sp
   // ▐[▌1⅓ sp
   // ▐]▌1⅓ sp
   // ▐:▌1⅓ sp
   // ▐:▌1⅓ sp
   // ▐(▌1⅓ sp
   // ▐)▌1⅓ sp
   // ▐{▌1⅔ sp
   // ▐}▌1⅔ sp
   // ▐"▌1⅔ sp
   // ▐?▌1⅔ sp
   // ▐<▌2 sp
   // ▐>▌2 sp
   // ▐^▌2 sp
   // ▐_▌2 sp
   // ▐~▌2 sp
   // ▐=▌2⅓ sp
   // ▐$▌2⅓ sp
   // ▐*▌2⅓ sp
   // ▐+▌2⅓ sp
   // ▐`▌2⅓ sp
   // ▐&▌2⅔ sp
   // ▐#▌2⅔ sp
   // ▐%▌3 sp
   // ▐@▌3⅓ sp
   // Punctuation avg. 1 sp (based on comma, full stop and dash being the most common)
   // 
   // 
   // 
   // ▄▄▄▄▄▄▄▄▄▄▄▄▄▄▄▄▄▄▄▄▄▄▄▄▄▄▄▄▄▄▄▄▄▄▄▄▄▄▄▄▄▄▄▄
   // ALL OTHER WHITESPACE CHARACTERS
   // 
   // The other whitespace characters (Hair space, figure space &c.) are supported by the Siemens
   // font, but have the identical widths to those listed above. The full list is shown below:
   // 
   // ▐  ▌2 Em spaces
   // ▐    ▌4 En space      (1/2 em)
   // ▐      ▌6 Three per em     (1/3 em)
   // ▐        ▌8 Punctuation space (1/4 em)
   // ▐        ▌8 Normal space      (1/4 em)
   // ▐        ▌8 Four per em      (1/4 em)
   // ▐        ▌8 Figure space     (1/4 em)
   // ▐            ▌12 Six per em    (1/6 em)
   // ▐            ▌12 Hair space       (1/6 em)
   // 
   //                 ━━━  ⬙⬙⬙⬙⬙⬙  ━━━
   // 
   // 
   // ██████████████ █ █ █ █  END   █ █ █ █ ██████████████
END_REGION

REGION Network 19: OB1 NETWORK 1 — Project description
   // ▀▀▀▀▀▀▀▀▀▀▀▀▀▀▀▀▀▀▀▀▀▀▀▀▀▀▀▀▀▀▀▀▀▀▀▀▀▀▀▀▀▀▀▀
   // 
   // TITLE:    PS2001 — PRACTICAL SERIES AUTOMATION LIBRARY
   // 
   // ▄▄▄▄▄▄▄▄▄▄▄▄▄▄▄▄▄▄▄▄▄▄▄▄▄▄▄▄▄▄▄▄▄▄▄▄▄▄▄▄▄▄▄▄
   // 
   // 
   // ――――――――――――――――――――――――――――――――――
   // COPYRIGHT:       © 2020 Michael Gledhill
   //           Part of the Practical Series of Publications
   //           Published in the United Kingdom
   //           mg@practicalseries.com
   //           https://practicalseries.com
   // ――――――――――――――――――――――――――――――――――
   // CUSTOMER:       Practical Series of Publications (PSP)
   // 
   // PROJECT:      Practical Series Automation Library (PAL)
   // 
   // PROJECT NO.:       PS2001
   // ――――――――――――――――――――――――――――――――――
   // CONTROLLER:       CPU 1515-2PN/DP
   // 
   // CONTROLLER NAME:    CON100
   // 
   // IP ADDRESS:      192.168.001.100
   // ――――――――――――――――――――――――――――――――――
   // TIA PROJECT NAME:    PS2001-PAL-D0000
   // 
   // STATUS:        DEVELOPMENT
   // ――――――――――――――――――――――――――――――――――
   // PROTECTION:     To minimise the risk of inadvertent modification to 
   //           tested modules, certain blocks will be released for 
   //           use with “protected access” (referred to a “write 
   //           protection” in Siemens terminology), this allows the 
   //           block to be used normally, but prevents the block 
   //           being accidentally modified. 
   // 
   //           This is in accordance with the risk assessment given 
   //           in the Validation Plant (VP), Appendix A [Ref. 002].
   // 
   //           ┌─────────────────────┐
   //           │ THE WRITE PROTECTION PASSWORD IS: PS2001 │
   //           └─────────────────────┘
   // 
   // 
   // ▄▄▄▄▄▄▄▄▄▄▄▄▄▄▄▄▄▄▄▄▄▄▄▄▄▄▄▄▄▄▄▄▄▄▄▄▄▄▄▄▄▄▄▄
   // PROJECT OVERVIEW
   // 
   // 
   // The PAL is a library of software modules and templates that have been developed for the 
   // Siemens Simatic S7-1500 range of controllers (and to a lesser extent the S7-1200 range).
   // 
   // The full library and all necessary documentation is available from the Practical Series website:
   // 
   //      https://practicalseries.com/2001-pal/index.html
   // 
   // 
   // The PAL is configured and deployed using the Siemens Simatic TIA Portal programming 
   // environment.
   // 
   // The PAL software structure is designed such that it is applicable to virtually all industrial 
   // applications that can generally controlled by a programmable logic controller.
   // 
   // The PAL software being developed as part of this Project, is considered to be suitable for use in 
   // the following types of industries (this is not an exhaustive list):
   // 
   //    •   Water and waste water treatment
   //    •   Pharmaceutical and batch production
   //    •   Brewing and fermentation
   //    •   Chemical manufacturing
   //    •   Oil and gas systems
   //    •   Food and beverage production
   // 
   // Such applications can generally be thought of as processes that operate with a response time
   // of more than 100 ms. I.e. the system would not be expected to respond to some stimuli faster
   // than 100 ms. In practice, a Controller may (and usually will) respond faster than this; however, 
   // a response time of 100 ms is considered to be an acceptable limit for PLC control.
   // 
   // At its most basic level, the PAL will be a library of software modules that control the fundamental 
   // aspects of an industrial plant; such modules would for example read the value of an instrument, 
   // operate a valve or drive, perform a calculation &c.
   // 
   // Such software modules are referred to as standard modules, these are fixed modules that 
   // perform a particular function and are identical across all software installations.
   // 
   // The PAL also contains application specific modules; these contain software that is applicable 
   // to the plant being controlled.
   // 
   // The Practical Series Automation Library is freely available under the MIT Open Source licence 
   // (see below). Those who find it useful may, if they wish, make a donation to support the library. 
   // 
   // Donations can be made here:
   // 
   //      https://practicalseries.com/2001-pal/11-web/81-00-pay.html
   // 
   // The PAL contains fully deployable software that has been developed by the author in his 
   // profession as a chartered electrical engineer. It is currently in use on various live plants 
   // throughout the UK and in some other parts of the world. 
   // 
   // This software is suitable for controlling and automating most industrial applications (typical 
   // process applications). It is easy to use and configure, but does have a degree of practical 
   // complexity appropriate for the environments within which it is employed. It is heavily 
   // configurable, has various operating modes and is suitable for a multitude of industrial 
   // applications.
   // 
   // IF YOU DON’T UNDERSTAND IT, DON’T USE IT. IF YOU DO USE IT, YOU DO SO AT YOUR OWN RISK.
   // 
   //                ━━━   ⬙⬙⬙⬙⬙⬙   ━━━
   // 
   // ▄▄▄▄▄▄▄▄▄▄▄▄▄▄▄▄▄▄▄▄▄▄▄▄▄▄▄▄▄▄▄▄▄▄▄▄▄▄▄▄▄▄▄▄
   // DOCUMENT REFERENCES
   // 
   // 
   //  ――――――――――――――――――――――――――――――――――――――――――
   //  REF.     DOCUMENT NO.       TITLE
   //  ――――――――――――――――――――――――――――――――――――――――――
   //  001  PS2001-5-0101-001   Quality Plan (QP)
   //  002  PS2001-5-0121-002   Validation Plan (VP)
   //  003  PS2001-5-0131-003   Test Plan (TP)
   //  004  PS2001-5-1101-001   User requirements specification (URS)
   //  005  PS2001-5-1111-001   Requirement Traceability Matrix (RTM)
   //  006  PS2001-5-2101-001   Functional Specification (FS) 
   //  007  PS2001-5-2211-001   Hardware Design Specification (HDS)
   //  008  PS2001-5-2311-001   Software Design Specification (SDS)
   //  009  PS2001-5-2313-011   Style Guide (SG)
   //  010  PS2001-5-234101-001    ES/WDP Configuration Manual
   //  011  PS2001-5-2312-fcNo.    Software Module Design Specification (SMDS)
   //  012  PS2001-5-2301-001   Software Module Register (SMR)
   //  013  PS2001-5-2302-011   Software Control and Mechanism (SCM)
   //  014  PS2001-5-7111-001   User Guide (UG)
   //  ――――――――――――――――――――――――――――――――――――――――――
   // 
   //                ━━━   ⬙⬙⬙⬙⬙⬙   ━━━
   // 
   // 
   // ▄▄▄▄▄▄▄▄▄▄▄▄▄▄▄▄▄▄▄▄▄▄▄▄▄▄▄▄▄▄▄▄▄▄▄▄▄▄▄▄▄▄▄▄
   // COMPLETED MODULES 
   // 
   // 
   //  ――――――――――――――――――――-―-- STATIC DATA       ― DYNAMIC  DAT A   ―
   //  BLOCK     NAME         REVISION    UDT/DB    REVISION  UDT/DB    REVISION  
   //  ――――――――――――――――――――――――――――――――――――――――――
   //  FC01001 StdSysGlobalData      001.000   UT 01000   001.000-R UT 21000   001.000-R
   //                  2020-11-20   UT 01001   001.000-R UT 21000   001.000-R 
   //                           None           DB21000   001.000-R
   //  ――――――――――――――――――――――――――――――――――――――――――
   //  FC02001 StdInstAnalogRead    001.000   UT 02001   001.000-R UT 22001   001.000-R
   //                  2020-11-20   DB02001   001.000-R DB22001   001.000-R
   //  ――――――――――――――――――――――――――――――――――――――――――
   //  FC18001 StdSubScaleAI      001.000   None           None 
   //                  2020-12-09   None           None
   //  ――――――――――――――――――――――――――――――――――――――――――
   //  FC18151 StdSubTimeEventRTC   001.000   None           UT 38151   001.000-R
   //                  2020-11-20                  DB38151   001.000-R
   //  ――――――――――――――――――――――――――――――――――――――――――
   //  FC61000 DocGenExample     001.000   None           None 
   //                  2020-11-20   None           None          
   //  ――――――――――――――――――――――――――――――――――――――――――
   //  FC21000 AppSys          001.000   None           None 
   //                  2020-12-04   None           None          
   //  ――――――――――――――――――――――――――――――――――――――――――
   //  See Software Module Register [Ref. 012] for full details
   // 
   //                ━━━   ⬙⬙⬙⬙⬙⬙   ━━━
   // 
   // 
   // ▀▀▀▀▀▀▀▀▀▀▀▀▀▀▀▀▀▀▀▀▀▀▀▀▀▀▀▀▀▀▀▀▀▀▀▀▀▀▀▀▀▀▀▀
   // LICENCE AND CONTACT INFORMATION
   // 
   // This software and its associated documentation is made available under the MIT Licence:
   // 
   // ════════════════════════════════════════════
   // 
   // The MIT License (MIT)
   // 
   // Copyright © 2020 Michael Gledhill
   // 
   // Permission is hereby granted, free of charge, to any person obtaining a copy of this software 
   // and associated documentation files (the “Software”), to deal in the Software without restriction, 
   // including without limitation the rights to use, copy, modify, merge, publish, distribute, 
   // sublicense, and/or sell copies of the Software, and to permit persons to whom the Software is 
   // furnished to do so, subject to the following conditions: 
   // 
   // The above copyright notice and this permission notice shall be included in all copies or 
   // substantial portions of the Software.
   // 
   // THE SOFTWARE IS PROVIDED “AS IS”, WITHOUT WARRANTY OF ANY KIND, EXPRESS OR IMPLIED, 
   // INCLUDING BUT NOT LIMITED TO THE WARRANTIES OF MERCHANTABILITY, FITNESS FOR A 
   // PARTICULAR PURPOSE AND NON-INFRINGEMENT. IN NO EVENT SHALL THE AUTHORS OR COPYRIGHT 
   // HOLDERS BE LIABLE FOR ANY CLAIM, DAMAGES OR OTHER LIABILITY, WHETHER IN AN ACTION OF 
   // CONTRACT, TORT OR OTHERWISE, ARISING FROM, OUT OF OR IN CONNECTION WITH THE SOFTWARE 
   // OR THE USE OR OTHER DEALINGS IN THE SOFTWARE.
   // 
   // ════════════════════════════════════════════
   //                    ┌────────────┐
   // You can reach the author by email here:   │  mg@practicalseries.com  │
   //                    └────────────┘
   // Questions, corrections, constructive criticism and complaints (polite ones) are invited.
   // 
   // ▄▄▄▄▄▄▄▄▄▄▄▄▄▄▄▄▄▄▄▄▄▄▄▄▄▄▄▄▄▄▄▄▄▄▄▄▄▄▄▄▄▄▄▄
   // 
   //                ━━━   ⬙⬙⬙⬙⬙⬙   ━━━
   // 
   // 
   // ██████████████ █ █ █ █  END   █ █ █ █ ██████████████
END_REGION

REGION Network 20: OB1 NETWORK 2 — Current revision and modification history
   // ▄▄▄▄▄▄▄▄▄▄▄▄▄▄▄▄▄▄▄▄▄▄▄▄▄▄▄▄▄▄▄▄▄▄▄▄▄▄▄▄▄▄▄▄
   // MODIFICATION HISTORY 
   // 
   // 
   // This is a complete summary of all primary software modifications (commit points) made to this 
   // TIA Portal project (the latest commit tag is at the top of the list). 
   // 
   // The latest commit tag, author and the date of the revision are hardcoded into the Controller in 
   // this network (allowing revision data to be obtained directly from the Controller).
   // 
   // The development of the software project is stored and managed within the GIT Source Code 
   // Management system (a version control system or VCS) in conjunction with the GitHub online 
   // hosting system. The software in its entirety is available in the GitHub remote repository:
   // 
   //      https://github.com/practicalseries/PS2001-pal-software
   // 
   // This repository is public and can be freely “forked” (copied) and used under the MIT Licence.
   // The MIT Licence is reproduced in full in the previous network.
   // 
   //  ———————————————————————————————————————————
   //  DATE       COMMIT TAG     AUTHOR        REASON FOR MODIFICATION
   //  ———————————————————————————————————————————
   //  2021.05.18    D0006B-000.101   M. Gledhill      FC01001 — RELEASED FOR USE
   // 
   //  2021.02.02    D0002      M. Gledhill      Baseline build
   // 
   //  2021.02.02    D0001      M. Gledhill      Hardware build
   // 
   //  2021.02.02    D0000      M. Gledhill      Initial commit — repository created
   //  ———————————————————————————————————————————
   // 
   // 
   // ▄▄▄▄▄▄▄▄▄▄▄▄▄▄▄▄▄▄▄▄▄▄▄▄▄▄▄▄▄▄▄▄▄▄▄▄▄▄▄▄▄▄▄▄
   RUNG wire#powerrail
      I_Contact( #SYS_SIGNALS._False )
      wire#w1
      S_Move(in := 'PS2001', out => #revInfo.REV_BLOCK)
   END_RUNG
   RUNG wire#w1
      S_Move(in := '001.000-R', out => #revInfo.REV_NUMBER)
   END_RUNG
   RUNG wire#w1
      S_Move(in := '2020.10.20', out => #revInfo.REV_DATE)
   END_RUNG
   RUNG wire#w1
      S_Move(in := 'M. Gledhill', out => #revInfo.REV_AUTHOR)
   END_RUNG
   // the same network as SCL:
   IF NOT #SYS_SIGNALS._False THEN
       #revInfo.REV_BLOCK := 'PS2001';
       #revInfo.REV_NUMBER := '001.000-R';
       #revInfo.REV_DATE := '2020.10.20';
       #revInfo.REV_AUTHOR := 'M. Gledhill';
   END_IF;
END_REGION

REGION Network 21: Load the system RTC and store in local variable [typical network comment]
   // ▀▀▀▀▀▀▀▀▀▀▀▀▀▀▀▀▀▀▀▀▀▀▀▀▀▀▀▀▀▀▀▀▀▀▀▀▀▀▀▀▀▀▀▀
   // The system block RD_SYS_T reads the time of day, the date and the day of week from the system 
   // real time clock as a DTL (or Date_And_Time_Long) data type (one just being the shorthand 
   // notation of the other). The result is stored in a local variable for decoding.
   // 
   // The DTL data type stores the date and time information in 8 consecutive bytes in BCD format 
   // as follows:
   // 
   // 
   //  ――――――――――――――――――――――――――――――――――――――――――
   //  DATA         DESCRIPTION
   // 
   //  0          Dear        (00h-89h = 2000 to 2089)   (90h-99h = 1990 to 1999)
   //  1          Month      (00h-12h = Jan to Dec)
   //  2          Day       (01h-31h)
   //  3          Hour        (00h-23h)
   //  4          Minute        (00h-59h)
   //  5          Month      (00h-12h = Jan to Dec)
   //  6-7         Millisecond      Uses byte 6 and most significant 4 bits of byte 7)
   //  7          Day of Week    least significant 4 bits (1h-7h = Sun to Sat)
   //  ――――――――――――――――――――――――――――――――――――――――――
   // 
   // 
   // The local variable is of type DTL (Date_And_Time_Long), this is compatible with the DT output
   // from RD_SYST, but allows the individual elements of the DT structure to be accesses
   // individually as symbols.
   // 
   // Note:    The DTL format can store more information (it can for example handle years in the 
   //      range 1970 to 2262; however, it will still only store the data in the table above
   //      when used with RS_SYS_T. 
   // ▄▄▄▄▄▄▄▄▄▄▄▄▄▄▄▄▄▄▄▄▄▄▄▄▄▄▄▄▄▄▄▄▄▄▄▄▄▄▄▄▄▄▄▄
END_REGION

REGION Network 22: ██ STEP 03340 — DECLARATION (RUNNING) [sequence network comment]
   // ▀▀▀▀▀▀▀▀▀▀▀▀▀▀▀▀▀▀▀▀▀▀▀▀▀▀▀▀▀▀▀▀▀▀▀▀▀▀▀▀▀▀▀▀
   // 
   //  ███   ███   ███  █  █   ███  
   // █   █ █   █ █   █ █  █  █   █ 
   // █  ██     █     █ █  █  █  ██ 
   // █ █ █  ███   ███  █████ █ █ █ 
   // ██  █     █     █    █  ██  █ 
   // █   █ █   █ █   █    █  █   █ 
   //  ███   ███   ███     █   ███  
   // 
   // ▄▄▄▄▄▄▄▄▄▄▄▄▄▄▄▄▄▄▄▄▄▄▄▄▄▄▄▄▄▄▄▄▄▄▄▄▄▄▄▄▄▄▄▄
   // STEP DESCRIPTION
   // 
   // 
   // Open the dry air purge valve (SV4201), activate the operator prompt ABORT PURGE.
   // 
   // If the main chamber humidity level falls below the target value proceed to the next step.
   // 
   // If the operator presses the ABORT PURGE button proceed to step 03400.
   // 
   // 
   // 
   // ▄▄▄▄▄▄▄▄▄▄▄▄▄▄▄▄▄▄▄▄▄▄▄▄▄▄▄▄▄▄▄▄▄▄▄▄▄▄▄▄▄▄▄▄
   // STEP PHASE AND DELAY CONDITIONS
   // 
   // 
   //  ――――――――――――――――――――――――――――――――――――――――――
   //  PHASE         ACTION
   //  ――――――――――――――――――――――――――――――――――――――――――
   //  INITIALISING      Activate the ABORT PURGE enable signal
   // 
   //  PROCESSING    Open SV4201
   // 
   //  TERMINATING    Clear the ABORT PURGE enable signal and any ABORT PURGE pressed
   //           signal
   // 
   //  STEP DELAY      No delay
   //  ――――――――――――――――――――――――――――――――――――――――――
   // 
   // 
   // 
   // ▄▄▄▄▄▄▄▄▄▄▄▄▄▄▄▄▄▄▄▄▄▄▄▄▄▄▄▄▄▄▄▄▄▄▄▄▄▄▄▄▄▄▄▄
   // STEP TRANSITION CONDITIONS
   // 
   // 
   //  ――――――――――――――――――――――――――――――――――――――――――
   //  TRANSITION      TO STEP    TRANSITION CONDITIONS
   //  ――――――――――――――――――――――――――――――――――――――――――
   //  1.        03350      HIC001 ≤ HUMIDITY_LIMIT
   // 
   //  2.        03400      Operator has pressed ABORT PURGE button
   //  ――――――――――――――――――――――――――――――――――――――――――
   // 
   // 
   // ▄▄▄▄▄▄▄▄▄▄▄▄▄▄▄▄▄▄▄▄▄▄▄▄▄▄▄▄▄▄▄▄▄▄▄▄▄▄▄▄▄▄▄▄
END_REGION

REGION Network 23: STEP 03340 — ACTION (INITIALISE) [sequence network comment]
   // ▀▀▀▀▀▀▀▀▀▀▀▀▀▀▀▀▀▀▀▀▀▀▀▀▀▀▀▀▀▀▀▀▀▀▀▀▀▀▀▀▀▀▀▀
   // INITIALISE PHASE
   // 
   // Activate the ABORT PURGE enable signal
   // (this is a temporary signal passed to the handling DB at the end of the block)
   // ▄▄▄▄▄▄▄▄▄▄▄▄▄▄▄▄▄▄▄▄▄▄▄▄▄▄▄▄▄▄▄▄▄▄▄▄▄▄▄▄▄▄▄▄
END_REGION

REGION Network 24: STEP 03340 — TRANSITION 01 [sequence network comment]
   // ▀▀▀▀▀▀▀▀▀▀▀▀▀▀▀▀▀▀▀▀▀▀▀▀▀▀▀▀▀▀▀▀▀▀▀▀▀▀▀▀▀▀▀▀
   // TRANSITION CONDITION 01
   // 
   // Wait for humidity to reach target level HIC001 ≤ HUMIDITY_LIMIT
   // ▄▄▄▄▄▄▄▄▄▄▄▄▄▄▄▄▄▄▄▄▄▄▄▄▄▄▄▄▄▄▄▄▄▄▄▄▄▄▄▄▄▄▄▄
END_REGION

REGION Network 25: LICENCE AND CONTACT INFORMATION [final network]
   // ▀▀▀▀▀▀▀▀▀▀▀▀▀▀▀▀▀▀▀▀▀▀▀▀▀▀▀▀▀▀▀▀▀▀▀▀▀▀▀▀▀▀▀▀
   // LICENCE AND CONTACT INFORMATION
   // 
   // This software and its associated documentation is made available under the MIT Licence:
   // 
   // ════════════════════════════════════════════
   // 
   // The MIT License (MIT)
   // 
   // Copyright © 2020 Michael Gledhill
   // 
   // Permission is hereby granted, free of charge, to any person obtaining a copy of this software 
   // and associated documentation files (the “Software”), to deal in the Software without restriction, 
   // including without limitation the rights to use, copy, modify, merge, publish, distribute, 
   // sublicense, and/or sell copies of the Software, and to permit persons to whom the Software is 
   // furnished to do so, subject to the following conditions: 
   // 
   // The above copyright notice and this permission notice shall be included in all copies or 
   // substantial portions of the Software.
   // 
   // THE SOFTWARE IS PROVIDED “AS IS”, WITHOUT WARRANTY OF ANY KIND, EXPRESS OR IMPLIED, 
   // INCLUDING BUT NOT LIMITED TO THE WARRANTIES OF MERCHANTABILITY, FITNESS FOR A 
   // PARTICULAR PURPOSE AND NON-INFRINGEMENT. IN NO EVENT SHALL THE AUTHORS OR COPYRIGHT 
   // HOLDERS BE LIABLE FOR ANY CLAIM, DAMAGES OR OTHER LIABILITY, WHETHER IN AN ACTION OF 
   // CONTRACT, TORT OR OTHERWISE, ARISING FROM, OUT OF OR IN CONNECTION WITH THE SOFTWARE 
   // OR THE USE OR OTHER DEALINGS IN THE SOFTWARE.
   // 
   // ════════════════════════════════════════════
   //                    ┌────────────┐
   // You can reach the author by email here:   │  mg@practicalseries.com  │
   //                    └────────────┘
   // Questions, corrections, constructive criticism and complaints (polite ones) are invited.
   // 
   // ▄▄▄▄▄▄▄▄▄▄▄▄▄▄▄▄▄▄▄▄▄▄▄▄▄▄▄▄▄▄▄▄▄▄▄▄▄▄▄▄▄▄▄▄
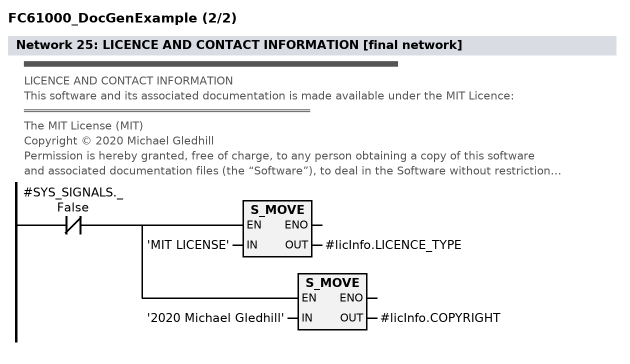
   RUNG wire#powerrail
      I_Contact( #SYS_SIGNALS._False )
      wire#w1
      S_Move(in := 'MIT LICENSE', out => #licInfo.LICENCE_TYPE)
   END_RUNG
   RUNG wire#w1
      S_Move(in := '2020 Michael Gledhill', out => #licInfo.COPYRIGHT)
   END_RUNG
   // the same network as SCL:
   IF NOT #SYS_SIGNALS._False THEN
       #licInfo.LICENCE_TYPE := 'MIT LICENSE';
       #licInfo.COPYRIGHT := '2020 Michael Gledhill';
   END_IF;
END_REGION
END_FUNCTION

FUNCTION "FC02001_StdInstAnalogRead" : Void   // FC2001, LAD
TITLE = Standard Module [INSTRUMENTATION] — Analog Instrument Read, Scale and Monitor
{ S7_Optimized_Access := 'TRUE' }
AUTHOR : M_Gledhill
FAMILY : Instrumentation
NAME : StdInstAnalogRead
VERSION : 2.8
// PRACTICAL SERIES AUTOMATION LIBRARY (PAL)   —   COPYRIGHT 2020 – M. GLEDHILL (MIT LICENCE)
//                   ———— ◆ ————
// FULL ONLINE DOCUMENTATION IS AVAILABLE AT: https://practicalseries.com/2001-pal/index.html
// stored: AutoNumber false, IsIECCheckEnabled true, SetENOAutomatically false, UDAEnableTagReadback false
   VAR_INPUT
      SYS_SIGNALS : "UT21000_Dy_SysSignals";   // Common system signals — logic and timing signals
      AI_RAW_SIGNAL : Int;   // Analog Input Signal
      AI_RAW_DATA : "UT00801_St_ConstAiRawData";   // Analog Input Signal — raw range and configuration data
      AI_SCALE_DATA : "UT00851_Sy_ConstAiScaleData";   // Analog Input Signal — scaled range and configuration data
      EXT_FAULT : Bool;   // Instrument External Fault (1 = Fault, 0 = Healthy)
   END_VAR
   VAR_IN_OUT
      STATIC_DATA : "UT02001_St_InstAnalogRead";   // Static data storage (UDT)
      DYNAMIC_DATA : "UT22001_Dy_InstAnalogRead";   // Dynamic data storage (UDT)
   END_VAR
   VAR_TEMP
      revInfo : "UT01000_St_SysRevision";   // Revision information for this block
      licInfo : "UT01001_St_SysLicence";   // Licence information for this block
      wrkAlmHEn : Bool;   // Working storage (Alm_H is enabled and not masked)
      wrkAlmLEn : Bool;   // Working storage (Alm_L is enabled and not masked)
      wrkWrnHEn : Bool;   // Working storage (Wrn_H is enabled and not masked)
      wrkWrnLEn : Bool;   // Working storage (Wrn_L is enabled and not masked)
      calPart1 : Real;   // Scale value calculation part 1 (RAW_ANALOG − RAW_MIN)
      calPart2 : Real;   // Scale value calculation part 2 (SCALE_MAX − SCALE_MIN)
      calPart3 : Real;   // Scale value calculation part 1 (RAW_MAX − RAW_MIN)
      calAbsOOR : Real;   // Calculated OOR absolute value in terms of the scaled value
      calHystAbs : Real;   // Absolute Hysteresis (in relation to alarm/warning)
      wrkHyst : Real;   // Working hysteresis value
      wrkOORPercent : Real;   // Working out of range percentage
      wrkInt : Int;   // Working storage (Integer)
      wrkReal : Real;   // Working storage (real)
      wrkDInt : DInt;   // Working storage (Double integer)
   END_VAR
   VAR_TEMP   // added for the SCL form of the ladder/FBD networks
      _w1 : Bool;
      _w2 : Bool;
      _w3 : Bool;
      _w4 : Bool;
   END_VAR
BEGIN

REGION Network 1: Block description — Sections 1 to 3.1
   // ▄▄▄▄▄▄▄▄▄▄▄▄▄▄▄▄▄▄▄▄▄▄▄▄▄▄▄▄▄▄▄▄▄  ＳＴＡＮＤＡＲＤ  ▄▄ 
   // 
   // 
   // TITLE:    INSTRUMENTATION — ANALOG INSTRUMENT READ, SCALE AND MONITOR
   // 
   // 
   // ▀▀▀▀▀▀▀▀▀▀▀▀▀▀▀▀▀▀▀▀▀▀▀▀▀▀▀▀▀▀▀▀▀▀▀▀▀▀▀▀▀▀▀▀ 
   // 
   // ┌──────────────────────────────────────────┐
   // │                                          │
   // │          FC02001 — SOFTWARE MODULE DESIGN SPECIFICATION (SMDS)            │
   // │                                          │
   // │      The PDF version of the SMDS for this module is available online here:        │
   // │              https://psop.uk/pal-smds-fc02001-p               │
   // │                                          │
   // │      It is also available as part of the Project User Defined Documentation,      │
   // │      it can be accessed by selecting this module in the Project Tree          │
   // │      (on the left) and pressing SHIFT+F1                        │
   // │                                          │
   // └─────────────────────────────────────── ʷᴵᴰ⁻ᵈᵉᵏ ┘
   // 
   // FC02001_StdInstAnalogRead reads and scales an analog instrument signal received via 
   // an analog input card.
   // 
   // The resultant scaled value is a real (floating point) number that matches the calibrated range of 
   // the instrument in engineering units.
   // 
   // The block has the facility to generate up to four alarms and warnings whenever the signal is 
   // beyond a specific setpoint value (either above or below); the four signals are:
   // 
   //    •   Alarm high
   // 
   //    •   Warning high
   // 
   //    •   Warning low
   // 
   //    •   Alarm low
   // 
   // Each alarm or warning can be time filtered (the condition must be present for a preset time 
   // before the alarm or warning is activated) and each will automatically reset when the signal is 
   // back within the acceptable range by a hysteresis amount.
   // 
   // In addition to the above four signals, various out-of-range fault signals will be generated if the 
   // instrument is outside its normal calibrated range by more than a specified percentage (this 
   // being a percentage of the total span of the instruments range).
   // 
   // The block can also generate an optional “external fault” signal from a hardwired fault input from 
   // the instrument itself.
   // 
   // The block has a simulation mode whereby the scaled value is replaced by an operator selected 
   // value (over-writing any signal from the instrument). This can be used for testing purposes or if 
   // the instrument is out of service for any reason.
   // 
   // 
   // 
   // 
   // 
   // ▄▄▄▄▄▄▄▄▄▄▄▄▄▄▄▄▄▄▄▄▄▄▄▄▄▄▄▄▄▄▄▄▄▄▄▄▄▄▄▄▄▄▄▄
   // 1.     BLOCK TECHNICAL SUMMARY
   // 
   // 
   //  ――――――――――――――――――――――――――――――――――――――――――
   //  NOMENCLATURE & ADDRESSING
   //  ――――――――――――――――――――――――――――――――――――――――――
   //  BLOCK TITLE         Analog Instrument Read, Scale and Alarm Monitoring
   //  BLOCK FUNCTION GROUP    Instrument 
   //  BLOCK ADDRESS       FC02001
   //  BLOCK SYMBOL        FC02001_StdInstAnalogRead
   //  BLOCK USER ID         StdInstAnalogRead
   // 
   //  ――――――――――――――――――――――――――――――――――――――――――
   //  BLOCK TYPE & USAGE
   //  ――――――――――――――――――――――――――――――――――――――――――
   //  BLOCK TYPE         Function (FC)
   //  BLOCK NUMBER        02001
   //  LANGUAGE           LAD
   //  OPTIMISED ACCESS     Yes
   //  PAL USAGE TYPE       Standard block
   // 
   //  ――――――――――――――――――――――――――――――――――――――――――
   //  METRICS
   //  ――――――――――――――――――――――――――――――――――――――――――
   //  EXECUTION TIME       87.7 μs¹
   //  LOAD MEMORY       93.3 kB
   //  WORK MEMORY           2.3 kB  
   //  ――――――――――――――――――――――――――――――――――――――――――
   //                ¹ Measured on: CPU-1515-2PN (order no. 6ES7512-2AM02-0AB0) 
   //                             https://psop.uk/pal-ds-cpu1515
   // 
   // 
   // 
   // ▂▂▂▂▂▂▂▂▂▂▂▂▂▂▂▂▂▂▂▂▂▂▂▂▂▂▂▂▂▂▂▂▂▂▂▂▂▂▂▂▂▂▂▂
   // 1.1      Additional document references
   // 
   // 
   // In addition to the documents referenced in OB1 (section DOCUMENT REFERENCES), the 
   // following documents are associated with this module:
   // 
   // 
   //  ――――――――――――――――――――――――――――――――――――――――――
   //  REF.     DOCUMENT NO.       TITLE
   //  ――――――――――――――――――――――――――――――――――――――――――
   //  101  PS2001-5-2312-db00801   DB00801 (analog input raw data) SMDS
   //  102  PS2001-5-2312-db00851   DB00851 (analog input scale data) SMDS
   //  ――――――――――――――――――――――――――――――――――――――――――
   // 
   //                ━━━   ⬙⬙⬙⬙⬙⬙   ━━━
   // 
   // 
   // ▄▄▄▄▄▄▄▄▄▄▄▄▄▄▄▄▄▄▄▄▄▄▄▄▄▄▄▄▄▄▄▄▄▄▄▄▄▄▄▄▄▄▄▄
   // 2.     FUNCTIONAL DESCRIPTION
   // 
   // 
   // This block is a comprehensive block designed to read and scale an analog instrument; it 
   // provides the following broad functions:
   // 
   //    •   Read an analog input, convert it to a real number that represents the calibrated 
   //      range of the instrument in engineering units
   // 
   //    •   Generate high and low alarm and warning signals to indicate that the instrument is 
   //      above or below specific thresholds
   // 
   //    •   Generate fault signals if the instrument is out of range or is indicating a specific fault 
   //      condition
   // 
   //    •   Provide simulation capabilities for testing and fault handling situations
   // 
   //    •   Generates the status and message signals necessary for symbolic representation at 
   //      a supervisory system (SCADA or HMI)
   // 
   // 
   // 
   // ▂▂▂▂▂▂▂▂▂▂▂▂▂▂▂▂▂▂▂▂▂▂▂▂▂▂▂▂▂▂▂▂▂▂▂▂▂▂▂▂▂▂▂▂
   // 2.1     Read and scale and instrument signal
   // 
   // 
   // The principal function of the block is to read a raw integer signal from an analog instrument 
   // (in the form of an input word, IW), and convert it into a scaled, floating point (real) number that 
   // reflects the calibrated reading of the instrument in question.
   // 
   // For example, if a flow meter with a calibrated range of -100 l/s to +100 l/s provided a 4-20 mA 
   // signal to the PLC, then 4 mA would represent -100 l/s and 20 mA would represent +100 l/s.
   // 
   // A typical 4-20 mA analog input signal returns a raw value of 0 at 4 mA and 27648 at 20 mA. 
   // 
   // The block would return scaled values as follows (it would also return every value in between; five 
   // typical values have been shown):
   // 
   // 
   //  ――――――――――――――――――――――――――――――――――――――――――
   //  RAW_SIGNAL          RAW INTEGER VALUE        RETURNED SCALE VALUE
   //  ――――――――――――――――――――――――――――――――――――――――――
   //     4 mA                      0             -100 l/s
   //     8 mA               6912                   -50 l/s
   //   12 mA             13824                   0 l/s
   //   16 mA             20736              +50 l/s
   //   20 mA             27648            +100 l/s
   //  ――――――――――――――――――――――――――――――――――――――――――
   // 
   // 
   // 
   // ▂▂▂▂▂▂▂▂▂▂▂▂▂▂▂▂▂▂▂▂▂▂▂▂▂▂▂▂▂▂▂▂▂▂▂▂▂▂▂▂▂▂▂▂
   // 2.2     Alarms and warnings
   // 
   // 
   // The block provides four alarm/warning signals:
   // 
   // 
   //  ――――――――――――――――――――――――――――――――――――――――――
   //  ALARM/WARNING         FUNCTION
   //  ――――――――――――――――――――――――――――――――――――――――――
   //  Alarm high            Scaled signal is equal to or above a preset alarm high 
   //                threshold (setpoint)
   // 
   //  Warning high           Scaled signal is equal to or above a preset warning high
   //                threshold (setpoint)
   // 
   //  Warning low          Scaled signal is equal to or above a preset warning low
   //                threshold (setpoint)
   // 
   //  Alarm low              Scaled signal is equal to or above a preset alarm low
   //                threshold (setpoint)
   //  ――――――――――――――――――――――――――――――――――――――――――
   // 
   // 
   // Alarms and warnings are individually enabled and are individually configurable.
   // 
   // Each alarm or warning has a threshold value (the value at which it becomes active); high alarms 
   // and warnings are active when the instrument is at or above the threshold level, low alarms and 
   // warnings are active when the instrument is at or below the threshold level. 
   // 
   // Each alarm or warning also has a hysteresis value (the instrument must be inside the threshold 
   // value by at least the hysteresis amount before the alarm/warning is reset).
   // 
   // Alarms and warnings automatically reset once the instrument is inside the threshold value by at 
   // least the hysteresis value.
   // 
   // Each alarm or warning is equipped with on and off time filtering (to prevent nuisance triggering 
   // of alarms and warnings) where:
   // 
   // ON FILTERING:  Delays the activation of the alarm/warning (signal must
   //          be on for a time period before the block conditioned 
   //          signal is activated).
   // 
   // OFF FILTERING:    Delays the alarm/warning from going off (i.e. the 
   //          conditioned signal will remain on for a time period
   //          once the input is reset).
   // 
   // Each alarm and warning has its own configurable on and off filtering delays.
   // 
   // 
   // 
   // ▂▂▂▂▂▂▂▂▂▂▂▂▂▂▂▂▂▂▂▂▂▂▂▂▂▂▂▂▂▂▂▂▂▂▂▂▂▂▂▂▂▂▂▂
   // 2.3     Fault signals
   // 
   // 
   // The block is able to generate four fault signals:
   // 
   //    •   External fault
   //    •   Instrument is over-range
   //    •   Instrument is under-range
   //    •   Instrument is out-of-range (common signal)
   // 
   // The external fault is generated by a hardwired signal from the instrument that indicates the 
   // instrument itself is reporting a fault. External fault signals are common with certain types of 
   // instruments (mass flow meters &c.) and are used to indicate such things as medium not present 
   // (liquid flow meters) or calibration and maintenance issues (instrument requires calibrating or 
   // cleaning or some other form of servicing).
   // 
   // Over-range and under-range faults are generated if the instrument is reading outside its normal 
   // calibrated range. Over-range if the instrument is reading higher than its maximum permitted 
   // value and under-range if lower than its minimum permitted value.
   // 
   // The level at which the instrument is considered to be either over-range or under-range (out of 
   // range), is set as a percentage of the whole instrument range (the span or full-scale deflection).
   //  
   // In the example of § 2.1, the instrument had a range of -100 to +100 l/s, this is a total range of 
   // 200 l/s, if the out of range value were set at 2.5%, this would be 2.5% of 200 l/s or 5 l/s. Thus, the 
   // instrument would be over-range if it were reading above 105 l/s; it would be under-range below
   // -105 l/s.
   // 
   // The out-of-range fault signal is a common signal that activates if either the over-range or 
   // under-range signal is active. It indicates the instrument is either over-range or under-range, but 
   // doesn’t specify which.
   // 
   // 
   // 
   // ▂▂▂▂▂▂▂▂▂▂▂▂▂▂▂▂▂▂▂▂▂▂▂▂▂▂▂▂▂▂▂▂▂▂▂▂▂▂▂▂▂▂▂▂
   // 2.4     Operating modes
   // 
   // 
   // The block supports the following optional modes of operation:
   // 
   //    •   Simulation mode (allows the operator to override the current instrument reading 
   //      with a simulated value)
   // 
   //    •   Remote/local/all selection (allows control of the instrument to be restricted to a 
   //      specific SCADA/HMI device) 
   // 
   //    •   Faceplate disabled (disables all optional modes)
   // 
   // 
   // 
   // ▁▁▁▁▁▁▁▁▁▁▁▁▁▁▁▁▁▁▁▁▁▁▁▁▁▁▁▁▁▁▁▁▁▁▁▁▁▁▁▁▁▁▁▁
   // 2.4.1     Simulation mode
   // 
   // 
   // The instrument can be switched to a simulation mode, in which the actual reading from the 
   // instrument is replaced by a simulated value provided by the operator. Simulation mode can be 
   // used during testing and can also be applied in a process environment if a fault condition is 
   // detected within the instrument.
   // 
   // Simulation mode is a manual operation that can only be initiated by an operator.
   // 
   // 
   // 
   // ▁▁▁▁▁▁▁▁▁▁▁▁▁▁▁▁▁▁▁▁▁▁▁▁▁▁▁▁▁▁▁▁▁▁▁▁▁▁▁▁▁▁▁▁
   // 2.4.2     Remote/local/all mode
   // 
   // 
   // Remote and local operating modes refer to the device that has control of the instrument; where 
   // a plant has more than one SCADA/HMI, say a SCADA in a remote control room and a field 
   // mounted HMI local to the instrument, it is possible to restrict the control of the instrument to 
   // one, or the other, or both devices as follows:
   // 
   //    •   Remote Only the remote system in the control room can control the device
   // 
   //    •   Local     A local system has taken control of the device and the remote system can 
   //            no longer issue commands to it
   // 
   //    •    All    Any system can control the device
   // 
   // The default arrangement is for all system to have access to the device.
   // 
   // 
   // 
   // ▁▁▁▁▁▁▁▁▁▁▁▁▁▁▁▁▁▁▁▁▁▁▁▁▁▁▁▁▁▁▁▁▁▁▁▁▁▁▁▁▁▁▁▁
   // 2.4.3     Faceplate disabled mode
   // 
   // 
   // Prevents the supervisory system from displaying the faceplate from which the above options are 
   // selected. If the faceplate is disabled, this module will set remote/local mode to ALL and will 
   // disable simulation mode.
   // 
   // 
   // 
   // ▁▁▁▁▁▁▁▁▁▁▁▁▁▁▁▁▁▁▁▁▁▁▁▁▁▁▁▁▁▁▁▁▁▁▁▁▁▁▁▁▁▁▁▁
   // 2.5      Supervisory system interface
   // 
   // 
   // See the online documentation for this block — select the block in the project tree and press:
   //      SHIFT + F1 or follow the link: https://psop.uk/pal-smds-fc02001-p 
   // 
   // The supervisory system interface is available in sections 2.5 and 4 of the online SMDS 
   // document.
   // 
   //                ━━━   ⬙⬙⬙⬙⬙⬙   ━━━
   // 
   // 
   // 
   // ▄▄▄▄▄▄▄▄▄▄▄▄▄▄▄▄▄▄▄▄▄▄▄▄▄▄▄▄▄▄▄▄▄▄▄▄▄▄▄▄▄▄▄▄
   // 3.     DETAILED BLOCK DESCRIPTION
   // 
   // 
   // This block, FC02001_StdInstAnalogRead uses user data types (UDTs)to provide the primary 
   // interface to the block. There are five formal parameters: 
   // 
   // 
   //  ――――――――――――――――――――――――――――――――――――――――――
   //  PARAM         FUNCTION                      TYPE      IN-OUT 
   //  ――――――――――――――――――――――――――――――――――――――――――
   //  SYS_SIGNALS      Common system signals                UT21000    In
   //           logic and timing signals for parametric access
   // 
   //  AI_RAW_SIGNAL      The unscaled analog input (input word          Word     In
   //           address for the IO card to which the instrument 
   //           is connected)
   //  AI_RAW_DATA      Analog input signal configuration data (type,     UT00801    In
   //           range, descriptions card parameters and 
   //           coefficients)
   // 
   //  AI_SCALE_DATA     Analog input signal scaled value data (instrument   UT00851   In
   //           tag, range, descriptions and engineering units)
   // 
   // 
   //  EXT_FAULT     Optional external fault signal for the instrument     Bool      In
   //           (1 = fault, 0 = healthy). If not required, set 
   //           permanently to _False
   // 
   //  STATIC_DATA     Data structure that holds the configuration data    UT02001    In
   //           for the instrument (raw range, scaled range 
   //           alarm and warning values, filtering times, 
   //           hysteresis values &c.)
   // 
   //  DYNAMIC_DATA      Data structure that holds the live data for the      UT22001    InOut
   //           instrument (its reading in engineering units, 
   //           any alarms or warnings that may be active, 
   //           current timer values, selected operating 
   //           mode &c.)
   //  ――――――――――――――――――――――――――――――――――――――――――
   // 
   // 
   // AI_RAW_SIGNAL and EXT_FAULT are signals provided directly from the instrument itself (via 
   // input cards). The AI_RAW_DATA and AI_SCALE_DATA parameters are UDTs that hold information 
   // about the nature of the AI_RAW_SIGNAL, in the case of AI_RAW_DATA its input type: voltage, 
   // current &c., its range in integer values and various parametric information and a textual 
   // description of the signal. In the case of AI_SCALE_DATA the scaled range of the signal, its 
   // engineering units, a textual description of the instrument and the instrument tag itself.
   // 
   // 
   //  ――――――――――――――――――――――――――――――――――――――――――
   //  PARAM         ASSOCIATED UDT            ASSOCIATED DATA BLOCK
   //  ――――――――――――――――――――――――――――――――――――――――――
   //  AI_RAW_DATA      UT00801_St_ConstAiRawData       DB00801_St_ConstAiRawData
   //  AI_SCALE_DATA     UT00851_St_ConstAiScaleData       DB00851_St_ConstAiScaleData
   //  ――――――――――――――――――――――――――――――――――――――――――
   // 
   // Section 3.1.1 contains a full description of the AI_RAW_DATA and AI_SCALE_DATA parameters
   // 
   // The other two parameters: STATIC_DATA and DYNAMIC_DATA are UDTs that hold (respectively) 
   // the configuration information and the live data for the instrument.
   // 
   // 
   //  ――――――――――――――――――――――――――――――――――――――――――
   //  PARAM         ASSOCIATED UDT            ASSOCIATED DATA BLOCK
   //  ――――――――――――――――――――――――――――――――――――――――――
   //  STATIC_DATA     UT02001_St_InstAnalogRead     DB02001_St_InstAnalogRead
   //  DYNAMIC_DATA      UT22001_Dy_InstAnalogRead       DB22001_Dy_InstAnalogRead
   //  ――――――――――――――――――――――――――――――――――――――――――
   // 
   // Section 6 contains a full list of all variables within these UDTs.
   // 
   // This arrangement conforms with the PAL philosophy whereby IO card connections have unique 
   // formal parameters; all remaining signals are passed as variables within UDTs.
   // 
   // 
   // 
   // ▂▂▂▂▂▂▂▂▂▂▂▂▂▂▂▂▂▂▂▂▂▂▂▂▂▂▂▂▂▂▂▂▂▂▂▂▂▂▂▂▂▂▂▂
   // 3.1     Converting the raw instrument signal to a scaled value
   // 
   // 
   // The AI_RAW_SIGNAL is the raw instrument signal received from an analog input card; this has 
   // specific ranges depending on the type of IO card and the type of signal in use.
   //  
   // Note:    It is assumed that the instrument has a linear response.
   // 
   // The following table shows example ranges for the AI_RAW_SIGNAL signal:
   // 
   //  ―――――――――――――――――――――――――――――――――――――――――― 
   //             LOWER LIMIT    EQUIVALENT UPPER LIMIT   EQUIVALENT
   //  SIGNAL TYPE      (RAW_MIN)         TO    (RAW_MAX)       TO      
   //  ―――――――――――――――――――――――――――――――――――――――――― 
   //  -10 V to 10 V         -27648     -10 V        27648      +10 V      
   //  1 V to 5 V          0      +1 V        27648     +5 V      
   //  -20 mA to 20 mA       -27648     -20 mA    27648      +20 mA      
   //  0 mA to 20 mA         0        0 mA    27648      +20 mA      
   //  4 mA to 20 mA (2w)      0        4 mA    27648      +20 mA      
   //  4 mA to 20 mA (4w)      0        4 mA    27648      +20 mA      
   //  RTD 150 Ω            0        0 Ω       27648      150 Ω      
   //  RTD 300 Ω            0        0 Ω       27648      300 Ω      
   //  PT x00           -2000       200.0°C      8500      850.0°C     
   //  Ni x00          -600     -60.0°C        250      250.0°C     
   //  Type B thermocouple     -2100      -210.0°C      12000    1200.0°C     
   //  Type K thermocouple     -2700      -270.0°C      13720    1372.0°C     
   //  ――――――――――――――――――――――――――――――――――――――――――
   //  Input ranges for typical instrument types (resistance thermometers and thermocouples)
   // 
   // 
   // The RAW_MIN and the RAW_MAX values in the above tables are the numerical values for the 
   // instrument range; the appropriate values are supplied as the RAW_MIN and RAW_MAX variables 
   // provided in the UDT of parameter AI_RAW_DATA. (see § 3.1.1 for a full description).
   // 	
   // 
   // The corresponding values for the scaled instrument signal are similarly provided by the 
   // SCALE_MIN and SCALE_MAX values provided in the UDT of parameter AI_SCALE_DATA. 
   // (see § 3.1.1for a full description).
   // 
   // Thus, if a flow meter with a calibrated range of –100 l/s to +100 l/s provided a 4-20 mA signal 
   // to the PLC, 
   // 
   // 
   //  ――――――――――――――――――――――――――――――――――――――――――
   //  SIGNAL NAME          FUNCTION                   VALUE
   //  ――――――――――――――――――――――――――――――――――――――――――
   //  AI_RAW_DATA.RAW_MIN     RANGE — Minimum value of the raw analog      0
   //                     signal (at the card)
   //  AI_RAW_DATA.RAW_MAX    RANGE — Maximum value of the raw analog        27648
   //                     signal (at the card)
   //  AI_SCALE_DATA.SCALE_MIN   RANGE — Minimum value of the scaled analog       -100 l/s
   //                     signal [engineering units]
   //  AI_SCALE_DATA.SCALE_MAX  RANGE — Maximum value of the scaled analog      +100 l/s
   //                     signal [engineering units]
   //  ――――――――――――――――――――――――――――――――――――――――――
   // 
   // The scaled value is stored in the DATA_DYNAMIC structure in the following variable:
   // 
   // 
   //  UT22001_Dy_InstAnalogRead
   //  ――――――――――――――――――――――――――――――――――――――――――
   //  SIGNAL NAME          FUNCTION                     TYPE
   //  ――――――――――――――――――――――――――――――――――――――――――
   //  actual_Value          ACTUAL — SCALED INSTRUMENT VALUE         Real
   //                      [engineering units]
   //  ――――――――――――――――――――――――――――――――――――――――――
   // 
   // 
   // The scaled value (actual_Value) is calculated as follows:
   // 
   // 
   // ┌─────────────────────────────────────────┐
   // │                              (AI_RAW_SIGNAL ─ RAW_MIN) ╳ (SCALE_MAX ─ SCALE_MIN)        │
   // │actual_Value =  ――――――――――――――――――――――――――  ┼ SCALE_MIN    │
   // │                              (RAW_MAX ─ RAW_MIN)                    │
   // └───────────────────────────────────  (3.1)  ───┘
   // Note:    RAW_MIN, RAW_MAX,  SCALE_MIN and SCALE_MAX are all preceded with RANGE_
   //      in the above equation 
   // 
   // 
   // 
   //            SCALE_VALUE
   //             ↑                    ⋰
   //            SCALE_MAX__│______________________________________⋰
   //             │                  ╱|
   //             │                 ╱ |     
   //             │                ╱  |
   //             │               ╱   |
   //             │              ╱    |
   //             │             ╱     |
   //             │            ╱      |
   //         actual_Value │<- - - - - - - - - - - - - - - - - - - - - ╱       |
   //             │          ╱ ⌃           |
   //             │         ╱ ╎       |
   //             │        ╱  ╎       |
   //             │       ╱   ╎       |   
   //             │      ╱    ╎       |
   //             │     ╱     ╎       |
   //             │    ╱         ╎          |
   //             SCALE_MIN__│______╱          ╎          |
   //             │  ⋰|           ╎          |
   //             │ ⋰ |           ╎          |
   //             ┼─────────────────────────→ AI_RAW_SIGNAL
   //                   |           ╎           |
   //                RAW_MIN        ╎        RAW_MAX
   //                       AI_RAW_SIGNAL
   // 
   //            Linear relationship between AI_RAW_SIGNAL and actual_Value
   // 
   // 
   // 
   // ▁▁▁▁▁▁▁▁▁▁▁▁▁▁▁▁▁▁▁▁▁▁▁▁▁▁▁▁▁▁▁▁▁▁▁▁▁▁▁▁▁▁▁▁
   // 3.1.1     Using AI_RAW_DATA and AI_SCALE_DATA
   // 
   // 
   // ▁▁▁▁▁▁▁▁▁▁▁▁▁▁▁▁▁▁▁▁▁▁▁▁▁▁▁▁▁▁▁▁▁▁▁▁▁▁▁▁▁▁▁▁
   // The AI_RAW_DATA parameter
   // 
   // The parameter AI_RAW_DATA is used to pass the analog input card type, range, description and
   // coefficient data used by all analog input card channels. Data is supplied to this parameter using
   // DB00801_St_ConstAiRawData, this contains a formal set of data for every type of Siemens 
   // analog input (datasets), E.g.: for a 4-wire 4-20 mA signal it is:
   // 
   //  AI_RAW_2003     "UT00801_St_ConstAiRawData" AI Current - 4-wire (4 mA to 20 mA)
   //   revInfo          "UT01000_St_SysRevision"
   //   ___________0010_0  Bool     false	 
   //   ___________0010_1  Bool     false
   //   AI_CODE       UInt      16#2003
   //   ___________0020_0  Bool     false
   //   ___________0020_1  Bool     false
   //   RAW_MIN          Int        0
   //   RAW_MAX         Int        27648
   //   RAW_DESC       String[60]    'Current - 4-wire (4 mA to 20 mA)'
   //   ___________0030_1  Bool     false
   //   ___________0030_2  Bool     false
   //   PARAM_TYPE       Byte        16#02
   //   PARAM_RANGE      Byte        16#03
   //   PARAM_COEF        Byte        16#00
   //   ___________0040_1  Bool     false
   //   ___________0040_2  Bool     false
   //   VALUE_COEF        Real        0.0
   // 
   // A full description of DB00801_St_ConstAiRawData and its associated datasets is given in 
   // [Ref. 101].
   // 
   // The whole dataset provided to the module via AI_RAW_DATA is copied to the DYNAMIC_DATA 
   // structure in the following variable:
   // 
   // 
   //  UT22001_Dy_InstAnalogRead
   //  ――――――――――――――――――――――――――――――――――――――――――
   //  SIGNAL NAME          FUNCTION                     TYPE
   //  ――――――――――――――――――――――――――――――――――――――――――
   //  actual_AiRawData       ACTUAL — A copy of the analog input AI_RAW_DATA     UT00801
   //                      parameter information
   //  ――――――――――――――――――――――――――――――――――――――――――
   // 
   // The primary in formation needed by the module are maximum and minimum ranges for the 
   // input signal, this information is given in in the DYNAMIC_DATA variables:
   // 
   // 
   //  UT22001_Dy_InstAnalogRead
   //  ――――――――――――――――――――――――――――――――――――――――――
   //  SIGNAL NAME           FUNCTION                    TYPE
   //  ――――――――――――――――――――――――――――――――――――――――――
   //  actual_AiRawData.RAW_MIN   ACTUAL — Minimum value of the analog input      Int
   //                       range being used by the module
   //  actual_AiRawData.RAW_MAX  ACTUAL — Maximum value of the analog input      Int
   //                       range being used by the module
   //  ――――――――――――――――――――――――――――――――――――――――――
   // 
   // These are the RAW_MIN and RAW_MAX values used in (3.1).
   // 
   // 
   // 
   // ▁▁▁▁▁▁▁▁▁▁▁▁▁▁▁▁▁▁▁▁▁▁▁▁▁▁▁▁▁▁▁▁▁▁▁▁▁▁▁▁▁▁▁▁
   // The AI_SCALE_DATA parameter
   // 
   // 
   // The AI_SCALE_DATA parameter is similar to the AI_RAW_DATA parameter except that in this case
   // it holds the scaled range, instrument tag, signal description and as-sociated engineering unit 
   // information. Data is supplied to this parameter using DB00851_St_ConstAiScaleData, this 
   // contains a set of data each instrument config-ured for the project, each instrument being a 
   // dataset. E.g.
   // 
   //  AI_SCALE_FC001   "UT00851_Sy_ConstAiScaleData"	
   //   revInfo        "UT01000_St_SysRevision"	
   //   ___________0010_0  Bool     false
   //   ___________0010_1  Bool     false
   //   AI_TAG           String[20]    'FC001'
   //   ___________0020_0  Bool     false
   //   ___________0020_1  Bool     false
   //   SCALE_MIN         Real        0.0
   //   SCALE_MAX        Real        1000.0
   //   SCALE_UNITS     String[20]    'l/s'
   //   SCALE_DESC      String[60]    'Inlet flow (0 to 1000 l/s)'
   // 
   // 
   // A full description of DB00851_St_ConstAiScaleData and its application is given in [Ref. 102].
   // 
   // The whole dataset provided to the module via AI_SCALE_DATA is copied to the DYNAMIC_DATA 
   // structure in the following variable:
   // 
   //  UT22001_Dy_InstAnalogRead
   //  ――――――――――――――――――――――――――――――――――――――――――
   //  SIGNAL NAME          FUNCTION                      TYPE
   //  ――――――――――――――――――――――――――――――――――――――――――
   //  actual_AiScaleData       FACTUAL — A copy of the analog input AI_SCALE_DATA UT00851
   //                      parameter information
   //  ――――――――――――――――――――――――――――――――――――――――――
   // 
   // The primary in formation needed by the module are maximum and minimum ranges for the 
   // scaled signal, this information is given in in the DYNAMIC_DATA variables
   // 
   // 
   //  UT22001_Dy_InstAnalogRead
   //  ――――――――――――――――――――――――――――――――――――――――――
   //  SIGNAL NAME            FUNCTION                    TYPE
   //  ――――――――――――――――――――――――――――――――――――――――――
   //  actual_AiScaleData.SCALE_MIN   ACTUAL — Minimum value of the analog input      Int
   //                        range being used by the module
   //  actual_AiScaleData.SCALE_MAX  ACTUAL — Maximum value of the analog input      Int
   //                        range being used by the module
   //  ――――――――――――――――――――――――――――――――――――――――――
   // 
   // These are the SCALE_MIN and SCALE_MAX values used in (3.1).
   // 
   // 
   // 
   // ▁▁▁▁▁▁▁▁▁▁▁▁▁▁▁▁▁▁▁▁▁▁▁▁▁▁▁▁▁▁▁▁▁▁▁▁▁▁▁▁▁▁▁▁
   // User defined analog input raw ranges
   // 
   // 
   // DB00801_St_ConstAiRawData contains a full set of analog card input ranges available to all 
   // Siemens Simatic analog input cards. However, if some non-Simatic card is being used 
   // (i.e. a third-party card that may have a Profinet or ProfiBus interface) it may be necessary to 
   // configure user defined RAW_MIN and RAW_MAX values. The module can accommodate this via the 
   // use of the AI_RAW_0000 dataset defined in data block DB00801_St_ConstAiRawData. Applying this
   // dataset to the AI_RAW_DATA parameter will cause the module to overwrite the 
   // actual_AiRawData.RAW_MIN and actual_AiRawData.RAW_MAX with data from the STATIC_DATA UDT 
   // parameter information. This contains the following:
   // 
   // 
   //  UT02001_St_InstAnalogRead
   //  ――――――――――――――――――――――――――――――――――――――――――
   //  SIGNAL NAME          FUNCTION                     TYPE
   //  ――――――――――――――――――――――――――――――――――――――――――
   //  RANGE_RAW_MIN       Optional minimum value of the raw analog signal	   Real
   //                (at the card). Only used if AI_RAW_DATA is set to 
   //                User Defined input (AI_RAW_0000)
   // 
   //  RANGE_RAW_MAX      Optional maximum value of the raw analog signal	   Real
   //               (at the card). Only used if AI_RAW_DATA is set to 
   //               User Defined input (AI_RAW_0000)
   //  ――――――――――――――――――――――――――――――――――――――――――
   // 
   // Note:    Only the RAW_MIN and RAW_MAX values are overwritten, the rest of the data in 
   //      actual_AiRawData is taken from the supplied AI_RAW_DATA dataset.
   // 
   // 
   // ████████████████████████████████████████████
   // █                                          █
   // █ RANGE_RAW_MIN and RANGE_RAW_MAX are only used if AI_RAW_DATA is set to the manual    █
   // █ configuration structure AI_RAW_0000.                         █
   // █                                          █
   // ████████████████████████████████████████████
   // 
   // 
   // 
   // ▁▁▁▁▁▁▁▁▁▁▁▁▁▁▁▁▁▁▁▁▁▁▁▁▁▁▁▁▁▁▁▁▁▁▁▁▁▁▁▁▁▁▁▁
   // 3.1.2     Configuration errors
   // 
   // 
   // The block requires that both the raw and scale range signals conform to certain rules::
   // 
   //    1.  actual_AiRawData.RAW_MIN must be less than, and not equal to 
   //      actual_AiRawData.RAW_MAX 
   // 
   //    2.  actual_AiScaleData.SCALE_MIN must be less than, and not equal to  
   //      actual_AiScaleData.SCALE_MIN
   // 
   // Should either of these conditions not be met, the signal: status_ConfigError will be activated 
   // (set true), additionally the three out of range signals (see § 3.4.1):
   // 
   //      msg_Flt_OverRange
   //      msg_Flt_UnderRange
   //      msg_Flt_OutOfRange
   // 
   // Will all be activated (this condition cannot be over-ridden by simulation mode, see § 3.4.1) and 
   // the actual_Value will be set to zero irrespective of any values given to AI_RAW_SIGNAL.
   // 
   // Note:    This avoids the potential for a divide by zero error: if the RAW_MIN and 
   //      RAW_MAX are exactly equal, the calculation of the actual_Value in 
   //      equation (3.1) would result in a divide by zero error.
END_REGION

